KUKA KRL program: MyProgram_208().src

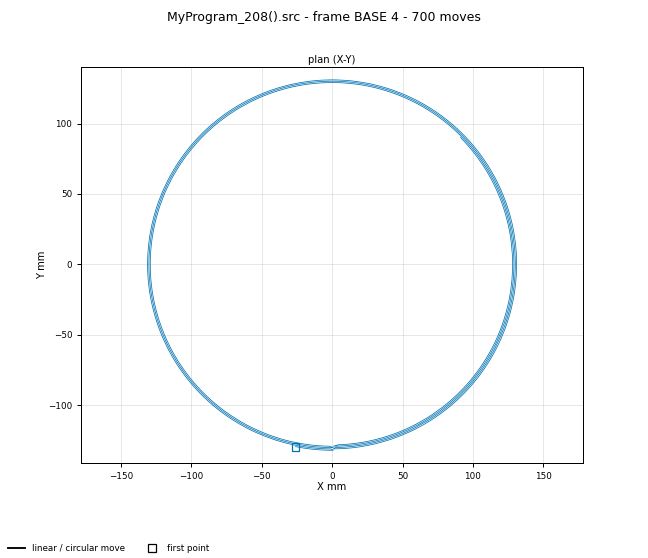
[picture p0: tool path of MyProgram_208().src in frame BASE 4, 700 of 700 moves have a stored position in this frame; points joined in program order, loops and branches not executed]
&ACCESS RVP
&REL 1
&PARAM TEMPLATE = C:\KRC\Roboter\Template\vorgabe
&PARAM EDITMASK = *
DEF MyProgram_208()
; ---- Setting reference (Base) ----
$BASE = BASE_DATA[4]

; --------------------------
; ---- Setting tool (TCP) ----
$TOOL = TOOL_DATA[3]
; --------------------------

$VEL.CP = VEL_APROX_PRINT
Startdeposition()
$VEL.CP = VEL_PRINT
LIN {X -25.9826,Y -129.3712,Z 148,A -104.0355,B 24.9663,C -1.3419,E1 24.9702,E2 190.502} C_DIS
LIN {X -21.9988,Y -130.1078,Z 148,A -102.3686,B 24.9665,C -1.3366,E1 24.9747,E2 188.8461} C_DIS
LIN {X -18.4843,Y -130.6533,Z 148,A -100.8231,B 24.9665,C -1.3362,E1 24.979,E2 187.3001} C_DIS
LIN {X -14.4168,Y -131.1647,Z 148,A -99.072,B 24.9666,C -1.3344,E1 24.9838,E2 185.5521} C_DIS
LIN {X -11.0414,Y -131.4916,Z 148,A -97.5626,B 24.9666,C -1.3363,E1 24.988,E2 184.0376} C_DIS
LIN {X -6.8374,Y -131.7773,Z 148,A -95.7546,B 24.9666,C -1.3352,E1 24.9931,E2 182.2315} C_DIS
LIN {X -3.1641,Y -131.9174,Z 148,A -94.0531,B 24.9663,C -1.3409,E1 24.9979,E2 180.5163} C_DIS
LIN {X 0.9361,Y -131.9509,Z 148,A -93.0717,B 24.9684,C -1.2997,E1 25.0004,E2 179.6325} C_DIS
Enddeposition()
LIN {X 0.9361,Y -131.9509,Z 148,A -93.0717,B 24.9684,C -1.2997,E1 25.0004,E2 179.6325} C_DIS
Startdeposition()
$VEL.CP = VEL_PRINT
LIN {X -0.9099,Y -130.9994,Z 148,A -93.7427,B 24.7462,C -1.2766,E1 24.7754,E2 180.3292} C_DIS
LIN {X -4.2416,Y -130.9351,Z 148,A -95.3676,B 24.7466,C -1.2679,E1 24.7708,E2 181.9751} C_DIS
LIN {X -8.0621,Y -130.754,Z 148,A -96.9489,B 24.7464,C -1.2724,E1 24.7664,E2 183.546} C_DIS
LIN {X -11.7713,Y -130.4745,Z 148,A -98.5272,B 24.7463,C -1.2749,E1 24.7621,E2 185.1191} C_DIS
LIN {X -15.6524,Y -130.0639,Z 148,A -100.2514,B 24.7463,C -1.2743,E1 24.7573,E2 186.8457} C_DIS
LIN {X -18.8652,Y -129.6372,Z 148,A -101.6954,B 24.7463,C -1.2733,E1 24.7533,E2 188.2933} C_DIS
LIN {X -23.4306,Y -128.8903,Z 148,A -103.7209,B 24.7463,C -1.2739,E1 24.7477,E2 190.3196} C_DIS
LIN {X -26.5584,Y -128.2825,Z 148,A -105.065,B 24.7462,C -1.2769,E1 24.744,E2 191.6579} C_DIS
LIN {X -29.9352,Y -127.5384,Z 148,A -106.5997,B 24.7462,C -1.2765,E1 24.7398,E2 193.1955} C_DIS
LIN {X -32.6648,Y -126.8651,Z 148,A -107.8332,B 24.7462,C -1.2771,E1 24.7365,E2 194.4294} C_DIS
LIN {X -35.721,Y -126.0387,Z 148,A -109.2219,B 24.7462,C -1.2778,E1 24.7328,E2 195.8187} C_DIS
LIN {X -38.4449,Y -125.2339,Z 148,A -110.4824,B 24.7462,C -1.2778,E1 24.7294,E2 197.0813} C_DIS
LIN {X -41.7109,Y -124.1847,Z 148,A -111.9951,B 24.7462,C -1.2784,E1 24.7254,E2 198.5953} C_DIS
LIN {X -44.8677,Y -123.0797,Z 148,A -113.4445,B 24.746,C -1.2804,E1 24.7216,E2 200.0429} C_DIS
LIN {X -47.7748,Y -121.9803,Z 148,A -114.8123,B 24.746,C -1.2813,E1 24.718,E2 201.4115} C_DIS
LIN {X -51.0457,Y -120.6491,Z 148,A -116.3473,B 24.7459,C -1.2833,E1 24.714,E2 202.9451} C_DIS
LIN {X -53.8492,Y -119.4232,Z 148,A -117.6982,B 24.7459,C -1.2842,E1 24.7106,E2 204.2971} C_DIS
LIN {X -56.7591,Y -118.0677,Z 148,A -119.1224,B 24.7458,C -1.2849,E1 24.707,E2 205.7232} C_DIS
LIN {X -59.8552,Y -116.5292,Z 148,A -120.6231,B 24.7457,C -1.2874,E1 24.7032,E2 207.2221} C_DIS
LIN {X -62.9418,Y -114.8929,Z 148,A -122.1788,B 24.7457,C -1.2881,E1 24.6994,E2 208.7805} C_DIS
LIN {X -66.1217,Y -113.0928,Z 148,A -123.8872,B 24.7457,C -1.285,E1 24.6953,E2 210.5014} C_DIS
LIN {X -70.1036,Y -110.6685,Z 148,A -125.8821,B 24.7455,C -1.2903,E1 24.6905,E2 212.4899} C_DIS
LIN {X -73.782,Y -108.2515,Z 148,A -127.8213,B 24.7455,C -1.2928,E1 24.686,E2 214.4298} C_DIS
LIN {X -77.2207,Y -105.8259,Z 148,A -129.6872,B 24.7453,C -1.2948,E1 24.6818,E2 216.2975} C_DIS
LIN {X -80.6432,Y -103.2414,Z 148,A -131.5951,B 24.7453,C -1.2966,E1 24.6776,E2 218.2079} C_DIS
LIN {X -84.0166,Y -100.515,Z 148,A -133.4733,B 24.745,C -1.3012,E1 24.6735,E2 220.0824} C_DIS
LIN {X -87.2683,Y -97.705,Z 148,A -135.3719,B 24.7449,C -1.304,E1 24.6695,E2 221.9817} C_DIS
LIN {X -90.6534,Y -94.5727,Z 148,A -137.3709,B 24.7446,C -1.3091,E1 24.6655,E2 223.9768} C_DIS
LIN {X -93.6988,Y -91.5564,Z 148,A -139.1989,B 24.7443,C -1.3154,E1 24.6619,E2 225.7975} C_DIS
LIN {X -96.2825,Y -88.8354,Z 148,A -140.9202,B 24.7443,C -1.3153,E1 24.6586,E2 227.5267} C_DIS
LIN {X -98.9862,Y -85.8131,Z 148,A -142.7358,B 24.7442,C -1.3174,E1 24.6552,E2 229.3455} C_DIS
LIN {X -101.8189,Y -82.4315,Z 148,A -144.6409,B 24.7439,C -1.3232,E1 24.6519,E2 231.2456} C_DIS
LIN {X -104.4895,Y -79.0187,Z 148,A -146.5452,B 24.7437,C -1.3275,E1 24.6486,E2 233.1489} C_DIS
LIN {X -107.1639,Y -75.352,Z 148,A -148.5233,B 24.7434,C -1.3328,E1 24.6454,E2 235.1238} C_DIS
LIN {X -109.6501,Y -71.6869,Z 148,A -150.5262,B 24.7434,C -1.3348,E1 24.6423,E2 237.1321} C_DIS
LIN {X -111.9772,Y -67.9938,Z 148,A -152.4303,B 24.743,C -1.3401,E1 24.6395,E2 239.0332} C_DIS
LIN {X -114.2442,Y -64.1113,Z 148,A -154.3647,B 24.7427,C -1.347,E1 24.6368,E2 240.9611} C_DIS
LIN {X -116.3464,Y -60.213,Z 148,A -156.2318,B 24.7422,C -1.3558,E1 24.6344,E2 242.8173} C_DIS
LIN {X -117.7191,Y -57.4802,Z 148,A -157.5744,B 24.7421,C -1.3594,E1 24.6327,E2 244.1586} C_DIS
LIN {X -119.1027,Y -54.555,Z 148,A -158.9968,B 24.7419,C -1.3631,E1 24.6311,E2 245.5798} C_DIS
LIN {X -120.3978,Y -51.6334,Z 148,A -160.4149,B 24.7417,C -1.3663,E1 24.6295,E2 246.9983} C_DIS
LIN {X -121.6766,Y -48.5441,Z 148,A -161.8738,B 24.7415,C -1.3708,E1 24.6279,E2 248.4546} C_DIS
LIN {X -122.8151,Y -45.5864,Z 148,A -163.2705,B 24.7413,C -1.3744,E1 24.6266,E2 249.8505} C_DIS
LIN {X -123.9258,Y -42.4751,Z 148,A -164.6967,B 24.741,C -1.3797,E1 24.6252,E2 251.2723} C_DIS
LIN {X -124.9291,Y -39.4266,Z 148,A -166.1227,B 24.7408,C -1.3829,E1 24.624,E2 252.6987} C_DIS
LIN {X -125.7713,Y -36.6488,Z 148,A -167.4085,B 24.7407,C -1.3861,E1 24.623,E2 253.9843} C_DIS
LIN {X -126.592,Y -33.7048,Z 148,A -168.7593,B 24.7405,C -1.3896,E1 24.622,E2 255.3347} C_DIS
LIN {X -127.3797,Y -30.5936,Z 148,A -170.171,B 24.7403,C -1.3936,E1 24.6211,E2 256.745} C_DIS
LIN {X -128.107,Y -27.3901,Z 148,A -171.6235,B 24.7401,C -1.3975,E1 24.6202,E2 258.1969} C_DIS
LIN {X -128.7553,Y -24.1625,Z 148,A -173.1573,B 24.7401,C -1.3976,E1 24.6194,E2 259.7394} C_DIS
LIN {X -129.4372,Y -20.1891,Z 148,A -174.8662,B 24.7396,C -1.4059,E1 24.6186,E2 261.4389} C_DIS
LIN {X -129.923,Y -16.7824,Z 148,A -176.3647,B 24.7394,C -1.411,E1 24.618,E2 262.9341} C_DIS
LIN {X -130.331,Y -13.2664,Z 148,A -177.8982,B 24.739,C -1.4167,E1 24.6176,E2 264.4631} C_DIS
LIN {X -130.5736,Y -10.5988,Z 148,A -179.0975,B 24.739,C -1.4192,E1 24.6173,E2 265.6636} C_DIS
LIN {X -130.8584,Y -6.1548,Z 148,A 178.9451,B 24.7386,C -1.4252,E1 24.617,E2 267.6187} C_DIS
LIN {X -130.9711,Y -2.9451,Z 148,A 177.3953,B 24.7387,C -1.423,E1 24.6168,E2 269.1831} C_DIS
LIN {X -131.002,Y 0.7144,Z 148,A 175.8358,B 24.7383,C -1.4302,E1 24.6168,E2 270.7349} C_DIS
LIN {X -130.9337,Y 4.2929,Z 148,A 174.3806,B 24.7378,C -1.4404,E1 24.6169,E2 272.1742} C_DIS
LIN {X -130.8001,Y 7.3151,Z 148,A 173.0287,B 24.7376,C -1.4434,E1 24.6171,E2 273.5272} C_DIS
LIN {X -130.6235,Y 9.9641,Z 148,A 171.835,B 24.7375,C -1.4458,E1 24.6174,E2 274.7225} C_DIS
LIN {X -130.3616,Y 12.9475,Z 148,A 170.5349,B 24.7372,C -1.4506,E1 24.6177,E2 276.0189} C_DIS
LIN {X -129.9903,Y 16.2694,Z 148,A 169.0609,B 24.737,C -1.4548,E1 24.6182,E2 277.4918} C_DIS
LIN {X -129.6518,Y 18.7633,Z 148,A 167.8956,B 24.737,C -1.4554,E1 24.6186,E2 278.6625} C_DIS
LIN {X -129.0893,Y 22.3185,Z 148,A 166.3617,B 24.7366,C -1.4624,E1 24.6193,E2 280.1888} C_DIS
LIN {X -128.5265,Y 25.3597,Z 148,A 164.9976,B 24.7363,C -1.4663,E1 24.62,E2 281.5517} C_DIS
LIN {X -127.9573,Y 28.0834,Z 148,A 163.7659,B 24.7362,C -1.4696,E1 24.6208,E2 282.7828} C_DIS
LIN {X -127.2826,Y 30.9963,Z 148,A 162.4348,B 24.736,C -1.4728,E1 24.6216,E2 284.1141} C_DIS
LIN {X -126.4618,Y 34.1929,Z 148,A 160.9953,B 24.7357,C -1.4776,E1 24.6226,E2 285.5505} C_DIS
LIN {X -125.6529,Y 37.0533,Z 148,A 159.6666,B 24.7355,C -1.4805,E1 24.6237,E2 286.8801} C_DIS
LIN {X -124.7469,Y 39.9969,Z 148,A 158.3113,B 24.7353,C -1.4844,E1 24.6248,E2 288.2338} C_DIS
LIN {X -123.666,Y 43.2244,Z 148,A 156.8135,B 24.7351,C -1.4887,E1 24.6262,E2 289.7299} C_DIS
LIN {X -122.5921,Y 46.1816,Z 148,A 155.4164,B 24.7349,C -1.4921,E1 24.6275,E2 291.1269} C_DIS
LIN {X -121.1977,Y 49.732,Z 148,A 153.7572,B 24.7346,C -1.4977,E1 24.6292,E2 292.782} C_DIS
LIN {X -120.0733,Y 52.384,Z 148,A 152.4837,B 24.7344,C -1.501,E1 24.6306,E2 294.0546} C_DIS
LIN {X -118.56,Y 55.7287,Z 148,A 150.8699,B 24.7341,C -1.5055,E1 24.6325,E2 295.6666} C_DIS
LIN {X -117.3472,Y 58.2341,Z 148,A 149.5948,B 24.7341,C -1.5066,E1 24.6341,E2 296.946} C_DIS
LIN {X -115.263,Y 62.2618,Z 148,A 147.5835,B 24.7338,C -1.5112,E1 24.6367,E2 298.9571} C_DIS
LIN {X -113.1673,Y 65.9948,Z 148,A 145.6202,B 24.7338,C -1.5125,E1 24.6394,E2 300.9276} C_DIS
LIN {X -110.9102,Y 69.7206,Z 148,A 143.7212,B 24.7334,C -1.5183,E1 24.6422,E2 302.8225} C_DIS
LIN {X -108.5273,Y 73.3745,Z 148,A 141.8388,B 24.733,C -1.5249,E1 24.6451,E2 304.6984} C_DIS
LIN {X -105.9314,Y 77.0752,Z 148,A 139.8594,B 24.7327,C -1.5303,E1 24.6483,E2 306.6746} C_DIS
LIN {X -103.3053,Y 80.5614,Z 148,A 137.9087,B 24.7325,C -1.5336,E1 24.6516,E2 308.6269} C_DIS
LIN {X -100.5874,Y 83.9302,Z 148,A 135.9813,B 24.7323,C -1.537,E1 24.655,E2 310.555} C_DIS
LIN {X -97.988,Y 86.9505,Z 148,A 134.3289,B 24.7318,C -1.5458,E1 24.6581,E2 312.1939} C_DIS
LIN {X -95.4585,Y 89.7203,Z 148,A 132.6064,B 24.7318,C -1.5461,E1 24.6613,E2 313.9232} C_DIS
LIN {X -92.6341,Y 92.6341,Z 148,A 130.8693,B 24.7314,C -1.5523,E1 24.6647,E2 315.653} C_DIS
LIN {X -89.7203,Y 95.4585,Z 148,A 129.1108,B 24.7311,C -1.5574,E1 24.6683,E2 317.4067} C_DIS
LIN {X -86.6644,Y 98.241,Z 148,A 127.2293,B 24.7311,C -1.5581,E1 24.6722,E2 319.294} C_DIS
LIN {X -83.3657,Y 101.0555,Z 148,A 125.3837,B 24.7307,C -1.5648,E1 24.6761,E2 321.1307} C_DIS
LIN {X -80.063,Y 103.6917,Z 148,A 123.5555,B 24.7304,C -1.5698,E1 24.6801,E2 322.9537} C_DIS
LIN {X -77.0752,Y 105.9314,Z 148,A 121.8208,B 24.7304,C -1.5685,E1 24.684,E2 324.6979} C_DIS
LIN {X -73.6336,Y 108.3519,Z 148,A 119.9486,B 24.7304,C -1.5707,E1 24.6883,E2 326.5713} C_DIS
LIN {X -69.7206,Y 110.9102,Z 148,A 117.9462,B 24.73,C -1.5767,E1 24.693,E2 328.5658} C_DIS
LIN {X -66.0255,Y 113.1493,Z 148,A 116.0341,B 24.7298,C -1.5791,E1 24.6976,E2 330.478} C_DIS
LIN {X -62.3681,Y 115.2059,Z 148,A 114.1343,B 24.7298,C -1.5792,E1 24.7023,E2 332.383} C_DIS
LIN {X -59.0536,Y 116.9373,Z 148,A 112.6504,B 24.7292,C -1.5892,E1 24.7059,E2 333.8468} C_DIS
LIN {X -55.9395,Y 118.4593,Z 148,A 111.127,B 24.7291,C -1.5913,E1 24.7097,E2 335.3693} C_DIS
LIN {X -52.7398,Y 119.9194,Z 148,A 109.5781,B 24.729,C -1.5931,E1 24.7137,E2 336.9176} C_DIS
LIN {X -50.0533,Y 121.0636,Z 148,A 108.3172,B 24.7288,C -1.5958,E1 24.7169,E2 338.1751} C_DIS
LIN {X -47.1892,Y 122.2079,Z 148,A 106.9282,B 24.7288,C -1.5958,E1 24.7205,E2 339.5672} C_DIS
LIN {X -43.6723,Y 123.5107,Z 148,A 105.3041,B 24.7287,C -1.5986,E1 24.7248,E2 341.1878} C_DIS
LIN {X -40.6267,Y 124.5457,Z 148,A 103.8953,B 24.7286,C -1.6002,E1 24.7285,E2 342.5954} C_DIS
LIN {X -38.1676,Y 125.3188,Z 148,A 102.7699,B 24.7285,C -1.6017,E1 24.7315,E2 343.7192} C_DIS
LIN {X -35.1038,Y 126.2113,Z 148,A 101.3643,B 24.7285,C -1.6027,E1 24.7353,E2 345.1247} C_DIS
LIN {X -32.0077,Y 127.0319,Z 148,A 99.9579,B 24.7283,C -1.6039,E1 24.7391,E2 346.5303} C_DIS
LIN {X -28.7342,Y 127.8127,Z 148,A 98.5168,B 24.7282,C -1.6067,E1 24.743,E2 347.9665} C_DIS
LIN {X -25.3597,Y 128.5265,Z 148,A 96.986,B 24.7282,C -1.6069,E1 24.7472,E2 349.4987} C_DIS
LIN {X -22.5439,Y 129.049,Z 148,A 95.7399,B 24.7281,C -1.6082,E1 24.7506,E2 350.7431} C_DIS
LIN {X -19.6104,Y 129.5268,Z 148,A 94.412,B 24.7281,C -1.6077,E1 24.7543,E2 352.0732} C_DIS
LIN {X -16.5908,Y 129.9481,Z 148,A 93.1019,B 24.728,C -1.6097,E1 24.7579,E2 353.3796} C_DIS
LIN {X -14.0238,Y 130.2495,Z 148,A 91.9555,B 24.728,C -1.6096,E1 24.7611,E2 354.527} C_DIS
LIN {X -10.7428,Y 130.5614,Z 148,A 90.4887,B 24.728,C -1.609,E1 24.7652,E2 355.9959} C_DIS
LIN {X -6.8071,Y 130.8256,Z 148,A 88.7518,B 24.728,C -1.6091,E1 24.77,E2 357.7332} C_DIS
LIN {X -3.2198,Y 130.9635,Z 148,A 87.2292,B 24.7278,C -1.6119,E1 24.7742,E2 359.2492} C_DIS
LIN {X -0.4557,Y 131.0019,Z 148,A 85.8758,B 24.7283,C -1.6051,E1 24.7781,E2 360.619} C_DIS
LIN {X 3.6364,Y 130.9519,Z 148,A 84.2162,B 24.7279,C -1.6117,E1 24.7827,E2 362.2624} C_DIS
LIN {X 7.3151,Y 130.8001,Z 148,A 82.6242,B 24.7278,C -1.6127,E1 24.7871,E2 363.8517} C_DIS
LIN {X 10.2809,Y 130.6004,Z 148,A 81.1754,B 24.7283,C -1.6052,E1 24.7912,E2 365.3176} C_DIS
LIN {X 13.9697,Y 130.2553,Z 148,A 79.6586,B 24.728,C -1.6102,E1 24.7953,E2 366.8216} C_DIS
LIN {X 17.7767,Y 129.7927,Z 148,A 78.0192,B 24.7279,C -1.6117,E1 24.7999,E2 368.4561} C_DIS
LIN {X 22.0621,Y 129.1321,Z 148,A 76.1251,B 24.7279,C -1.6112,E1 24.8051,E2 370.3494} C_DIS
LIN {X 24.7907,Y 128.6352,Z 148,A 74.8752,B 24.728,C -1.6089,E1 24.8085,E2 371.6035} C_DIS
LIN {X 28.0834,Y 127.9573,Z 148,A 73.4127,B 24.728,C -1.6085,E1 24.8125,E2 373.0649} C_DIS
LIN {X 31.4626,Y 127.1702,Z 148,A 71.9179,B 24.728,C -1.6087,E1 24.8166,E2 374.557} C_DIS
LIN {X 34.1929,Y 126.4618,Z 148,A 70.7054,B 24.728,C -1.609,E1 24.8198,E2 375.7668} C_DIS
LIN {X 37.0053,Y 125.6669,Z 148,A 69.3938,B 24.7282,C -1.6064,E1 24.8234,E2 377.0824} C_DIS
LIN {X 40.1901,Y 124.6852,Z 148,A 67.9494,B 24.7282,C -1.6059,E1 24.8272,E2 378.5254} C_DIS
LIN {X 43.2147,Y 123.6694,Z 148,A 66.5628,B 24.7282,C -1.6052,E1 24.8309,E2 379.911} C_DIS
LIN {X 46.5227,Y 122.4644,Z 148,A 65.0073,B 24.7284,C -1.6028,E1 24.835,E2 381.4688} C_DIS
LIN {X 49.3702,Y 121.3436,Z 148,A 63.6779,B 24.7284,C -1.6019,E1 24.8384,E2 382.7973} C_DIS
LIN {X 52.7398,Y 119.9194,Z 148,A 62.0809,B 24.7286,C -1.6003,E1 24.8425,E2 384.3944} C_DIS
LIN {X 55.7287,Y 118.56,Z 148,A 60.6472,B 24.7286,C -1.5987,E1 24.8461,E2 385.8283} C_DIS
LIN {X 58.3798,Y 117.2754,Z 148,A 59.3607,B 24.7287,C -1.5971,E1 24.8494,E2 387.1149} C_DIS
LIN {X 61.3241,Y 115.763,Z 148,A 57.8918,B 24.7289,C -1.5941,E1 24.853,E2 388.5869} C_DIS
LIN {X 65.1192,Y 113.673,Z 148,A 55.9562,B 24.7292,C -1.5893,E1 24.8577,E2 390.5283} C_DIS
LIN {X 68.8477,Y 111.4547,Z 148,A 54.062,B 24.7294,C -1.5865,E1 24.8623,E2 392.423} C_DIS
LIN {X 72.3878,Y 109.1887,Z 148,A 52.2524,B 24.7294,C -1.585,E1 24.8665,E2 394.2303} C_DIS
LIN {X 75.8535,Y 106.8102,Z 148,A 50.467,B 24.7295,C -1.5846,E1 24.8706,E2 396.0105} C_DIS
LIN {X 79.0297,Y 104.4811,Z 148,A 48.712,B 24.7298,C -1.5798,E1 24.8745,E2 397.7705} C_DIS
LIN {X 82.2119,Y 101.996,Z 148,A 46.9168,B 24.7301,C -1.5749,E1 24.8785,E2 399.5705} C_DIS
LIN {X 85.6299,Y 99.144,Z 148,A 44.9716,B 24.7303,C -1.5712,E1 24.8826,E2 401.517} C_DIS
LIN {X 88.8354,Y 96.2825,Z 148,A 43.1745,B 24.7303,C -1.5716,E1 24.8863,E2 403.3058} C_DIS
LIN {X 91.6109,Y 93.6454,Z 148,A 41.4111,B 24.7308,C -1.5634,E1 24.8899,E2 405.0814} C_DIS
LIN {X 94.8522,Y 90.3609,Z 148,A 39.4288,B 24.7309,C -1.5608,E1 24.8937,E2 407.0614} C_DIS
LIN {X 97.7478,Y 87.2205,Z 148,A 37.5996,B 24.7311,C -1.5585,E1 24.8972,E2 408.8878} C_DIS
LIN {X 100.515,Y 84.0166,Z 148,A 35.7335,B 24.7314,C -1.5533,E1 24.9005,E2 410.7576} C_DIS
LIN {X 103.1734,Y 80.7298,Z 148,A 33.8816,B 24.7316,C -1.5486,E1 24.9038,E2 412.6119} C_DIS
LIN {X 105.8259,Y 77.2207,Z 148,A 31.917,B 24.732,C -1.5416,E1 24.907,E2 414.5836} C_DIS
LIN {X 108.3519,Y 73.6336,Z 148,A 30.0263,B 24.7322,C -1.5382,E1 24.9101,E2 416.4732} C_DIS
LIN {X 110.9102,Y 69.7206,Z 148,A 28.0434,B 24.7324,C -1.536,E1 24.913,E2 418.4512} C_DIS
LIN {X 113.1673,Y 65.9948,Z 148,A 26.1559,B 24.7326,C -1.5317,E1 24.9157,E2 420.3392} C_DIS
LIN {X 115.2059,Y 62.3681,Z 148,A 24.2716,B 24.7331,C -1.5232,E1 24.9183,E2 422.2337} C_DIS
LIN {X 117.0275,Y 58.8765,Z 148,A 22.6931,B 24.733,C -1.526,E1 24.9203,E2 423.7971} C_DIS
LIN {X 118.56,Y 55.7287,Z 148,A 21.1812,B 24.7332,C -1.5226,E1 24.9221,E2 425.309} C_DIS
LIN {X 119.6843,Y 53.2656,Z 148,A 20.0021,B 24.7333,C -1.5194,E1 24.9235,E2 426.4891} C_DIS
LIN {X 121.0636,Y 50.0533,Z 148,A 18.488,B 24.7335,C -1.5157,E1 24.9251,E2 428.0036} C_DIS
LIN {X 122.2269,Y 47.1405,Z 148,A 17.133,B 24.7337,C -1.5125,E1 24.9265,E2 429.3587} C_DIS
LIN {X 123.3409,Y 44.1432,Z 148,A 15.7214,B 24.734,C -1.5076,E1 24.9278,E2 430.774} C_DIS
LIN {X 124.3201,Y 41.3042,Z 148,A 14.4251,B 24.7342,C -1.5045,E1 24.929,E2 432.0702} C_DIS
LIN {X 125.3157,Y 38.1777,Z 148,A 12.9994,B 24.7344,C -1.5005,E1 24.9302,E2 433.497} C_DIS
LIN {X 126.2072,Y 35.1185,Z 148,A 11.6291,B 24.7346,C -1.4975,E1 24.9312,E2 434.8667} C_DIS
LIN {X 127.0727,Y 31.8469,Z 148,A 10.1551,B 24.7348,C -1.4931,E1 24.9323,E2 436.3425} C_DIS
LIN {X 127.8127,Y 28.7342,Z 148,A 8.7503,B 24.7351,C -1.4884,E1 24.9332,E2 437.7503} C_DIS
LIN {X 128.6645,Y 24.6376,Z 148,A 6.9511,B 24.7353,C -1.4842,E1 24.9341,E2 439.5487} C_DIS
LIN {X 129.2392,Y 21.42,Z 148,A 5.5014,B 24.7357,C -1.4786,E1 24.9348,E2 441.0034} C_DIS
LIN {X 129.7927,Y 17.7767,Z 148,A 3.942,B 24.7357,C -1.4761,E1 24.9355,E2 442.5593} C_DIS
LIN {X 130.106,Y 15.299,Z 148,A 2.8055,B 24.7361,C -1.4702,E1 24.9358,E2 443.7029} C_DIS
LIN {X 130.4745,Y 11.7713,Z 148,A 1.3213,B 24.7362,C -1.4687,E1 24.9362,E2 445.1818} C_DIS
LIN {X 130.7283,Y 8.4797,Z 148,A -0.2002,B 24.7367,C -1.4599,E1 24.9366,E2 446.7154} C_DIS
LIN {X 130.912,Y 4.872,Z 148,A -1.7245,B 24.7368,C -1.4577,E1 24.9367,E2 448.2357} C_DIS
LIN {X 131.002,Y 0.7144,Z 148,A -3.4745,B 24.7369,C -1.4554,E1 24.9368,E2 449.9806} C_DIS
LIN {X 130.9722,Y -2.9078,Z 148,A -5.2225,B 24.7377,C -1.4413,E1 24.9368,E2 451.7515} C_DIS
LIN {X 130.8339,Y -6.6416,Z 148,A -6.7322,B 24.7377,C -1.4426,E1 24.9366,E2 453.249} C_DIS
LIN {X 130.6236,Y -9.9637,Z 148,A -8.1088,B 24.7377,C -1.4421,E1 24.9363,E2 454.6186} C_DIS
LIN {X 130.3684,Y -12.8768,Z 148,A -9.4087,B 24.738,C -1.4367,E1 24.936,E2 455.9235} C_DIS
LIN {X 130.0947,Y -15.394,Z 148,A -10.5205,B 24.7382,C -1.4329,E1 24.9356,E2 457.0379} C_DIS
LIN {X 129.6895,Y -18.4992,Z 148,A -11.8686,B 24.7384,C -1.4295,E1 24.9351,E2 458.3859} C_DIS
LIN {X 129.2136,Y -21.5734,Z 148,A -13.2338,B 24.7386,C -1.4248,E1 24.9345,E2 459.7542} C_DIS
LIN {X 128.6271,Y -24.8331,Z 148,A -14.6845,B 24.7389,C -1.4199,E1 24.9337,E2 461.208} C_DIS
LIN {X 127.9742,Y -28.0053,Z 148,A -16.0595,B 24.739,C -1.4175,E1 24.933,E2 462.5806} C_DIS
LIN {X 127.3166,Y -30.8556,Z 148,A -17.3794,B 24.7393,C -1.4112,E1 24.9321,E2 463.9077} C_DIS
LIN {X 126.4618,Y -34.1929,Z 148,A -18.8401,B 24.7395,C -1.4087,E1 24.9311,E2 465.3657} C_DIS
LIN {X 125.5957,Y -37.2487,Z 148,A -20.2217,B 24.7397,C -1.4047,E1 24.93,E2 466.749} C_DIS
LIN {X 124.5457,Y -40.6267,Z 148,A -21.7601,B 24.7399,C -1.4001,E1 24.9287,E2 468.2894} C_DIS
LIN {X 123.6698,Y -43.2134,Z 148,A -22.9532,B 24.7401,C -1.3964,E1 24.9276,E2 469.4845} C_DIS
LIN {X 122.553,Y -46.2861,Z 148,A -24.4084,B 24.7404,C -1.3905,E1 24.9262,E2 470.9455} C_DIS
LIN {X 121.1977,Y -49.732,Z 148,A -25.9806,B 24.7406,C -1.388,E1 24.9246,E2 472.515} C_DIS
LIN {X 120.1282,Y -52.2569,Z 148,A -27.1936,B 24.7408,C -1.3835,E1 24.9232,E2 473.7318} C_DIS
LIN {X 118.56,Y -55.7287,Z 148,A -28.83,B 24.741,C -1.3799,E1 24.9213,E2 475.3679} C_DIS
LIN {X 117.2754,Y -58.3798,Z 148,A -30.1338,B 24.7412,C -1.3752,E1 24.9197,E2 476.6759} C_DIS
LIN {X 115.2492,Y -62.2875,Z 148,A -32.083,B 24.7416,C -1.3681,E1 24.9171,E2 478.6317} C_DIS
LIN {X 113.1673,Y -65.9948,Z 148,A -34.0125,B 24.7421,C -1.3588,E1 24.9145,E2 480.5731} C_DIS
LIN {X 110.9102,Y -69.7206,Z 148,A -35.8882,B 24.7423,C -1.3548,E1 24.9117,E2 482.4486} C_DIS
LIN {X 108.4477,Y -73.492,Z 148,A -37.7809,B 24.7423,C -1.3533,E1 24.9088,E2 484.3354} C_DIS
LIN {X 105.9314,Y -77.0752,Z 148,A -39.6338,B 24.7425,C -1.3512,E1 24.9058,E2 486.1842} C_DIS
LIN {X 103.9114,Y -79.7776,Z 148,A -41.1238,B 24.7427,C -1.3464,E1 24.9033,E2 487.6785} C_DIS
LIN {X 101.7057,Y -82.5719,Z 148,A -42.7689,B 24.7432,C -1.3374,E1 24.9004,E2 489.3371} C_DIS
LIN {X 98.8753,Y -85.9403,Z 148,A -44.6686,B 24.7434,C -1.3336,E1 24.8969,E2 491.2371} C_DIS
LIN {X 96.037,Y -89.1007,Z 148,A -46.5061,B 24.7436,C -1.3299,E1 24.8935,E2 493.0753} C_DIS
LIN {X 93.2317,Y -92.0327,Z 148,A -48.1771,B 24.7436,C -1.3309,E1 24.8902,E2 494.7366} C_DIS
LIN {X 90.3932,Y -94.8213,Z 148,A -49.9567,B 24.7438,C -1.3246,E1 24.8867,E2 496.5238} C_DIS
LIN {X 87.2205,Y -97.7478,Z 148,A -51.8564,B 24.7441,C -1.3194,E1 24.8827,E2 498.428} C_DIS
LIN {X 84.0166,Y -100.515,Z 148,A -53.6511,B 24.7441,C -1.3182,E1 24.8789,E2 500.2187} C_DIS
LIN {X 80.7537,Y -103.1546,Z 148,A -55.5423,B 24.7445,C -1.3111,E1 24.8748,E2 502.1195} C_DIS
LIN {X 77.2207,Y -105.8259,Z 148,A -57.5105,B 24.7448,C -1.3053,E1 24.8703,E2 504.0944} C_DIS
LIN {X 73.6336,Y -108.3519,Z 148,A -59.4103,B 24.7449,C -1.3024,E1 24.866,E2 505.9946} C_DIS
LIN {X 69.8274,Y -110.8429,Z 148,A -61.3616,B 24.745,C -1.3004,E1 24.8614,E2 507.9441} C_DIS
LIN {X 65.9948,Y -113.1673,Z 148,A -63.36,B 24.7453,C -1.2948,E1 24.8566,E2 509.9499} C_DIS
LIN {X 62.3681,Y -115.2059,Z 148,A -65.1704,B 24.7454,C -1.292,E1 24.8521,E2 511.7615} C_DIS
LIN {X 59.1648,Y -116.8807,Z 148,A -66.6277,B 24.7453,C -1.2958,E1 24.8486,E2 513.2058} C_DIS
LIN {X 55.7287,Y -118.56,Z 148,A -68.2736,B 24.7453,C -1.2944,E1 24.8444,E2 514.8506} C_DIS
LIN {X 52.961,Y -119.8205,Z 148,A -69.5912,B 24.7453,C -1.293,E1 24.8411,E2 516.1682} C_DIS
LIN {X 50.0533,Y -121.0636,Z 148,A -70.9749,B 24.7455,C -1.2909,E1 24.8375,E2 517.5535} C_DIS
LIN {X 47.0313,Y -122.2693,Z 148,A -72.3811,B 24.7455,C -1.2898,E1 24.8338,E2 518.9594} C_DIS
LIN {X 44.1233,Y -123.3481,Z 148,A -73.7456,B 24.7457,C -1.2875,E1 24.8303,E2 520.3263} C_DIS
LIN {X 41.1815,Y -124.361,Z 148,A -75.1282,B 24.7458,C -1.2847,E1 24.8266,E2 521.713} C_DIS
LIN {X 37.5745,Y -125.5003,Z 148,A -76.7467,B 24.7458,C -1.2845,E1 24.8223,E2 523.3289} C_DIS
LIN {X 34.9655,Y -126.25,Z 148,A -77.9362,B 24.7458,C -1.2831,E1 24.8191,E2 524.5198} C_DIS
LIN {X 31.7159,Y -127.106,Z 148,A -79.3886,B 24.7459,C -1.2825,E1 24.8151,E2 525.9715} C_DIS
LIN {X 28.0834,Y -127.9573,Z 148,A -81.0973,B 24.7462,C -1.2769,E1 24.8105,E2 527.691} C_DIS
LIN {X 24.6708,Y -128.6582,Z 148,A -82.5559,B 24.7461,C -1.279,E1 24.8065,E2 529.143} C_DIS
LIN {X 21.4033,Y -129.242,Z 148,A -84.0214,B 24.7461,C -1.2771,E1 24.8024,E2 530.6114} C_DIS
LIN {X 17.7767,Y -129.7927,Z 148,A -85.5848,B 24.7461,C -1.2781,E1 24.7981,E2 532.1711} C_DIS
LIN {X 14.446,Y -130.2041,Z 148,A -87.1273,B 24.7464,C -1.2734,E1 24.7938,E2 533.7236} C_DIS
LIN {X 10.9505,Y -130.5439,Z 148,A -88.6103,B 24.7463,C -1.2753,E1 24.7897,E2 535.2013} C_DIS
LIN {X 7.5386,Y -130.7863,Z 148,A -90.1836,B 24.7465,C -1.2706,E1 24.7853,E2 536.7849} C_DIS
LIN {X 3.6802,Y -130.9507,Z 148,A -91.8016,B 24.7463,C -1.2737,E1 24.7808,E2 538.3952} C_DIS
LIN {X 0.9276,Y -130.9972,Z 148,A -92.5799,B 24.7453,C -1.2951,E1 24.7788,E2 539.1223} C_DIS
Enddeposition()
LIN {X 0.9276,Y -130.9972,Z 148,A -92.5799,B 24.7453,C -1.2951,E1 24.7788,E2 539.1223} C_DIS
Startdeposition()
$VEL.CP = VEL_PRINT
LIN {X 2.2953,Y -130.0302,Z 148,A -91.3636,B 23.7072,C -1.1309,E1 23.737,E2 538.1694} C_DIS
LIN {X 6.6533,Y -129.8801,Z 148,A -89.594,B 23.7075,C -1.1242,E1 23.7419,E2 536.4172} C_DIS
LIN {X 9.7391,Y -129.6854,Z 148,A -88.0412,B 23.707,C -1.1341,E1 23.7462,E2 534.8404} C_DIS
LIN {X 15.3426,Y -129.1421,Z 148,A -85.4485,B 23.7067,C -1.1411,E1 23.7535,E2 532.2323} C_DIS
LIN {X 22.0886,Y -128.1621,Z 148,A -82.6745,B 23.7071,C -1.1319,E1 23.7611,E2 529.4839} C_DIS
LIN {X 24.9925,Y -127.6274,Z 148,A -81.1427,B 23.7066,C -1.1444,E1 23.7654,E2 527.9229} C_DIS
LIN {X 28.6488,Y -126.8557,Z 148,A -79.6943,B 23.7069,C -1.1361,E1 23.7692,E2 526.4972} C_DIS
LIN {X 32.1676,Y -126.0091,Z 148,A -78.1664,B 23.707,C -1.1344,E1 23.7734,E2 524.9759} C_DIS
LIN {X 35.2573,Y -125.1799,Z 148,A -76.7005,B 23.7068,C -1.1387,E1 23.7773,E2 523.5019} C_DIS
LIN {X 40.3053,Y -123.649,Z 148,A -74.4302,B 23.7068,C -1.1387,E1 23.7834,E2 521.2359} C_DIS
LIN {X 42.7685,Y -122.8165,Z 148,A -73.2712,B 23.7068,C -1.1409,E1 23.7864,E2 520.0739} C_DIS
LIN {X 46.2368,Y -121.5549,Z 148,A -71.1381,B 23.7054,C -1.1686,E1 23.7922,E2 517.877} C_DIS
LIN {X 50.1024,Y -120.0114,Z 148,A -69.7611,B 23.7064,C -1.1482,E1 23.7956,E2 516.5539} C_DIS
LIN {X 53.2812,Y -118.6344,Z 148,A -68.2432,B 23.7063,C -1.1501,E1 23.7995,E2 515.0352} C_DIS
LIN {X 56.4292,Y -117.1703,Z 148,A -66.7981,B 23.7063,C -1.1483,E1 23.8031,E2 513.5986} C_DIS
LIN {X 59.5458,Y -115.6185,Z 148,A -65.1445,B 23.706,C -1.1569,E1 23.8073,E2 511.9285} C_DIS
LIN {X 68.4575,Y -110.5763,Z 148,A -60.8352,B 23.706,C -1.1547,E1 23.8177,E2 507.6383} C_DIS
LIN {X 71.6464,Y -108.5371,Z 148,A -59.1404,B 23.7059,C -1.1594,E1 23.8216,E2 505.9379} C_DIS
LIN {X 73.7755,Y -107.1013,Z 148,A -57.8907,B 23.7055,C -1.1677,E1 23.8245,E2 504.6722} C_DIS
LIN {X 77.141,Y -104.7032,Z 148,A -56.0866,B 23.7054,C -1.1706,E1 23.8286,E2 502.8674} C_DIS
LIN {X 80.6325,Y -102.0392,Z 148,A -53.9414,B 23.7047,C -1.1856,E1 23.8334,E2 500.6936} C_DIS
LIN {X 84.5859,Y -98.7868,Z 148,A -51.9149,B 23.705,C -1.179,E1 23.8377,E2 498.6918} C_DIS
LIN {X 87.493,Y -96.2209,Z 148,A -50.2088,B 23.7048,C -1.1829,E1 23.8412,E2 496.9833} C_DIS
LIN {X 90.7138,Y -93.1912,Z 148,A -48.0833,B 23.7041,C -1.1967,E1 23.8456,E2 494.8329} C_DIS
LIN {X 95.3225,Y -88.4711,Z 148,A -45.4695,B 23.7045,C -1.1889,E1 23.8506,E2 492.2504} C_DIS
LIN {X 97.7461,Y -85.7864,Z 148,A -43.7702,B 23.704,C -1.1984,E1 23.8537,E2 490.5355} C_DIS
LIN {X 100.499,Y -82.544,Z 148,A -41.911,B 23.7038,C -1.2026,E1 23.8571,E2 488.6749} C_DIS
LIN {X 104.8446,Y -76.9485,Z 148,A -38.866,B 23.7036,C -1.2072,E1 23.8622,E2 485.634} C_DIS
LIN {X 107.2408,Y -73.5723,Z 148,A -36.9714,B 23.7032,C -1.2159,E1 23.8653,E2 483.7276} C_DIS
LIN {X 109.7634,Y -69.754,Z 148,A -34.9555,B 23.7029,C -1.2216,E1 23.8683,E2 481.7083} C_DIS
LIN {X 112.1721,Y -65.8095,Z 148,A -33.0092,B 23.7029,C -1.2229,E1 23.8711,E2 479.7694} C_DIS
LIN {X 114.3113,Y -62.0199,Z 148,A -31.067,B 23.7025,C -1.2299,E1 23.8738,E2 477.8207} C_DIS
LIN {X 115.9464,Y -58.9017,Z 148,A -28.4624,B 23.6995,C -1.2896,E1 23.8772,E2 475.083} C_DIS
LIN {X 119.1992,Y -52.0068,Z 148,A -25.8254,B 23.7009,C -1.262,E1 23.8801,E2 472.5297} C_DIS
LIN {X 120.7381,Y -48.3258,Z 148,A -24.6417,B 23.7021,C -1.2376,E1 23.8813,E2 471.4132} C_DIS
LIN {X 121.7721,Y -45.6569,Z 148,A -23.3042,B 23.7018,C -1.2455,E1 23.8826,E2 470.0641} C_DIS
LIN {X 122.8587,Y -42.6466,Z 148,A -21.8722,B 23.7015,C -1.2511,E1 23.8839,E2 468.6268} C_DIS
LIN {X 123.9362,Y -39.4062,Z 148,A -20.377,B 23.7013,C -1.2553,E1 23.8852,E2 467.1299} C_DIS
LIN {X 125.1218,Y -35.4647,Z 148,A -18.561,B 23.701,C -1.2613,E1 23.8866,E2 465.3104} C_DIS
LIN {X 126.0203,Y -32.1237,Z 148,A -17.0646,B 23.7008,C -1.2647,E1 23.8877,E2 463.8145} C_DIS
LIN {X 126.8016,Y -28.8859,Z 148,A -15.6363,B 23.7007,C -1.2674,E1 23.8886,E2 462.3884} C_DIS
LIN {X 127.7404,Y -24.4014,Z 148,A -13.5464,B 23.7001,C -1.2776,E1 23.8898,E2 460.2861} C_DIS
LIN {X 128.4897,Y -20.0868,Z 148,A -11.6788,B 23.7,C -1.2807,E1 23.8906,E2 458.4225} C_DIS
LIN {X 128.9973,Y -16.5203,Z 148,A -9.8632,B 23.6991,C -1.2977,E1 23.8913,E2 456.5761} C_DIS
LIN {X 129.5403,Y -11.5212,Z 148,A -7.8346,B 23.6992,C -1.2952,E1 23.8918,E2 454.5665} C_DIS
LIN {X 129.8602,Y -7.0499,Z 148,A -6.0844,B 23.6995,C -1.29,E1 23.8922,E2 452.8402} C_DIS
LIN {X 130.0292,Y -2.3595,Z 148,A -3.7403,B 23.6984,C -1.3111,E1 23.8924,E2 450.4587} C_DIS
LIN {X 130.045,Y 1.3751,Z 148,A -2.3098,B 23.6987,C -1.3053,E1 23.8924,E2 449.0516} C_DIS
LIN {X 129.9651,Y 4.7226,Z 148,A -0.8294,B 23.6985,C -1.3104,E1 23.8922,E2 447.5679} C_DIS
LIN {X 129.7939,Y 8.165,Z 148,A 0.7383,B 23.6981,C -1.3179,E1 23.892,E2 445.9916} C_DIS
LIN {X 129.305,Y 13.9025,Z 148,A 2.8947,B 23.6987,C -1.3064,E1 23.8915,E2 443.8772} C_DIS
LIN {X 128.4526,Y 20.3265,Z 148,A 6.0721,B 23.6973,C -1.3321,E1 23.8902,E2 440.656} C_DIS
LIN {X 127.8429,Y 23.8649,Z 148,A 7.9085,B 23.6963,C -1.3503,E1 23.8893,E2 438.786} C_DIS
LIN {X 127.02,Y 27.9137,Z 148,A 9.4046,B 23.6969,C -1.3392,E1 23.8884,E2 437.3265} C_DIS
LIN {X 126.3945,Y 30.6184,Z 148,A 10.6068,B 23.6968,C -1.342,E1 23.8877,E2 436.1249} C_DIS
LIN {X 125.6331,Y 33.6058,Z 148,A 11.9971,B 23.6965,C -1.3479,E1 23.8867,E2 434.7286} C_DIS
LIN {X 124.5943,Y 37.2809,Z 148,A 13.8105,B 23.6958,C -1.3598,E1 23.8852,E2 432.8968} C_DIS
LIN {X 123.4235,Y 40.9834,Z 148,A 15.3828,B 23.6959,C -1.3579,E1 23.8839,E2 431.3386} C_DIS
LIN {X 122.2954,Y 44.2361,Z 148,A 16.8735,B 23.6958,C -1.3611,E1 23.8825,E2 429.8488} C_DIS
LIN {X 120.9876,Y 47.7008,Z 148,A 19.1439,B 23.6937,C -1.3989,E1 23.8801,E2 427.4984} C_DIS
LIN {X 119.0594,Y 52.3283,Z 148,A 20.6469,B 23.6953,C -1.3689,E1 23.8785,E2 426.0782} C_DIS
LIN {X 117.4073,Y 55.9331,Z 148,A 22.1513,B 23.6957,C -1.3615,E1 23.8768,E2 424.6006} C_DIS
LIN {X 116.527,Y 57.7449,Z 148,A 23.2987,B 23.6949,C -1.3773,E1 23.8753,E2 423.4207} C_DIS
LIN {X 114.9731,Y 60.7806,Z 148,A 24.8278,B 23.6946,C -1.3829,E1 23.8734,E2 421.8864} C_DIS
LIN {X 112.8485,Y 64.6431,Z 148,A 27.4784,B 23.6922,C -1.4246,E1 23.8696,E2 419.1472} C_DIS
LIN {X 110.0125,Y 69.3594,Z 148,A 29.2375,B 23.6938,C -1.3968,E1 23.8671,E2 417.4662} C_DIS
LIN {X 107.5387,Y 73.1366,Z 148,A 31.2003,B 23.6936,C -1.4007,E1 23.8641,E2 415.5043} C_DIS
LIN {X 105.0513,Y 76.6671,Z 148,A 33.1462,B 23.6932,C -1.4077,E1 23.8609,E2 413.551} C_DIS
LIN {X 102.3407,Y 80.2487,Z 148,A 35.0574,B 23.6932,C -1.4091,E1 23.8576,E2 411.6458} C_DIS
LIN {X 99.555,Y 83.6796,Z 148,A 36.9948,B 23.6929,C -1.4133,E1 23.8542,E2 409.7075} C_DIS
LIN {X 96.6473,Y 87.0223,Z 148,A 39.4574,B 23.6912,C -1.4437,E1 23.8495,E2 407.1812} C_DIS
LIN {X 93.4223,Y 90.475,Z 148,A 40.8453,B 23.6929,C -1.4132,E1 23.847,E2 405.8753} C_DIS
LIN {X 90.842,Y 93.0661,Z 148,A 42.9214,B 23.6914,C -1.4401,E1 23.8427,E2 403.7418} C_DIS
LIN {X 88.1871,Y 95.5853,Z 148,A 44.155,B 23.6923,C -1.4243,E1 23.8403,E2 402.5525} C_DIS
LIN {X 85.4811,Y 98.0125,Z 148,A 45.8187,B 23.6919,C -1.4307,E1 23.8368,E2 400.8801} C_DIS
LIN {X 82.0334,Y 100.9163,Z 148,A 47.8151,B 23.6917,C -1.435,E1 23.8325,E2 398.881} C_DIS
LIN {X 78.5567,Y 103.6455,Z 148,A 49.7254,B 23.6916,C -1.4368,E1 23.8283,E2 396.9738} C_DIS
LIN {X 75.1686,Y 106.1283,Z 148,A 51.6047,B 23.6913,C -1.4415,E1 23.824,E2 395.0899} C_DIS
LIN {X 71.4553,Y 108.6628,Z 148,A 53.563,B 23.6912,C -1.4436,E1 23.8195,E2 393.1333} C_DIS
LIN {X 67.6252,Y 111.0875,Z 148,A 55.5833,B 23.6909,C -1.4479,E1 23.8147,E2 391.1092} C_DIS
LIN {X 63.7927,Y 113.3312,Z 148,A 57.4818,B 23.6909,C -1.4479,E1 23.8101,E2 389.2169} C_DIS
LIN {X 59.8603,Y 115.4563,Z 148,A 59.3477,B 23.6911,C -1.4454,E1 23.8055,E2 387.3625} C_DIS
LIN {X 57.4965,Y 116.6495,Z 148,A 60.513,B 23.691,C -1.4469,E1 23.8026,E2 386.1969} C_DIS
LIN {X 54.6446,Y 118.0125,Z 148,A 61.9197,B 23.6908,C -1.4493,E1 23.799,E2 384.7881} C_DIS
LIN {X 51.318,Y 119.497,Z 148,A 63.5134,B 23.6908,C -1.4506,E1 23.7949,E2 383.1954} C_DIS
LIN {X 48.0134,Y 120.8641,Z 148,A 65.3024,B 23.6901,C -1.4627,E1 23.7902,E2 381.3806} C_DIS
LIN {X 44.1092,Y 122.3412,Z 148,A 66.9275,B 23.6906,C -1.4539,E1 23.7861,E2 379.7808} C_DIS
LIN {X 40.9409,Y 123.4377,Z 148,A 68.3859,B 23.6906,C -1.4543,E1 23.7822,E2 378.3245} C_DIS
LIN {X 37.7146,Y 124.4618,Z 148,A 69.9072,B 23.6904,C -1.4569,E1 23.7781,E2 376.7996} C_DIS
LIN {X 33.7301,Y 125.6,Z 148,A 71.7538,B 23.6903,C -1.4592,E1 23.7732,E2 374.9506} C_DIS
LIN {X 29.982,Y 126.5479,Z 148,A 73.3656,B 23.6905,C -1.4558,E1 23.7688,E2 373.3498} C_DIS
LIN {X 27.2776,Y 127.1574,Z 148,A 74.6881,B 23.6901,C -1.4613,E1 23.7652,E2 372.0153} C_DIS
LIN {X 23.1182,Y 127.9791,Z 148,A 77.0053,B 23.6888,C -1.4839,E1 23.7587,E2 369.6448} C_DIS
LIN {X 18.8854,Y 128.6726,Z 148,A 78.4843,B 23.6899,C -1.4646,E1 23.7547,E2 368.2154} C_DIS
LIN {X 14.5056,Y 129.2401,Z 148,A 80.2388,B 23.6905,C -1.4558,E1 23.7499,E2 366.4842} C_DIS
LIN {X 8.07,Y 129.7998,Z 148,A 83.4088,B 23.6895,C -1.4715,E1 23.741,E2 363.2767} C_DIS
LIN {X 4.0818,Y 129.9872,Z 148,A 84.9941,B 23.69,C -1.4631,E1 23.7366,E2 361.7129} C_DIS
LIN {X 0.548,Y 130.0494,Z 148,A 86.5701,B 23.69,C -1.4637,E1 23.7322,E2 360.1354} C_DIS
LIN {X -5.1544,Y 129.9482,Z 148,A 89.0445,B 23.6901,C -1.4612,E1 23.7253,E2 357.6668} C_DIS
LIN {X -11.5584,Y 129.5371,Z 148,A 91.7441,B 23.6906,C -1.454,E1 23.7179,E2 354.9843} C_DIS
LIN {X -15.6756,Y 129.1024,Z 148,A 93.7157,B 23.6902,C -1.46,E1 23.7123,E2 352.9965} C_DIS
LIN {X -21.5546,Y 128.2516,Z 148,A 96.3552,B 23.6902,C -1.4593,E1 23.7051,E2 350.3563} C_DIS
LIN {X -24.9746,Y 127.6309,Z 148,A 97.786,B 23.6906,C -1.4533,E1 23.7012,E2 348.9386} C_DIS
LIN {X -28.4018,Y 126.9122,Z 148,A 99.4538,B 23.6903,C -1.4578,E1 23.6966,E2 347.2574} C_DIS
LIN {X -32.0276,Y 126.0447,Z 148,A 101.0035,B 23.6907,C -1.4519,E1 23.6924,E2 345.7202} C_DIS
LIN {X -35.2536,Y 125.1809,Z 148,A 102.4787,B 23.6907,C -1.4506,E1 23.6884,E2 344.2459} C_DIS
LIN {X -38.4131,Y 124.248,Z 148,A 104.2828,B 23.6899,C -1.4654,E1 23.6835,E2 342.4015} C_DIS
LIN {X -41.6499,Y 123.201,Z 148,A 105.4677,B 23.6909,C -1.449,E1 23.6805,E2 341.2553} C_DIS
LIN {X -45.8053,Y 121.7165,Z 148,A 107.3919,B 23.691,C -1.4456,E1 23.6755,E2 339.3355} C_DIS
LIN {X -48.989,Y 120.4708,Z 148,A 108.9911,B 23.691,C -1.4478,E1 23.6713,E2 337.727} C_DIS
LIN {X -52.3437,Y 119.0533,Z 148,A 110.5262,B 23.6912,C -1.4422,E1 23.6674,E2 336.202} C_DIS
LIN {X -54.7437,Y 117.9666,Z 148,A 111.6662,B 23.6914,C -1.4395,E1 23.6645,E2 335.0658} C_DIS
LIN {X -57.6898,Y 116.5542,Z 148,A 113.0943,B 23.6916,C -1.4367,E1 23.6609,E2 333.6407} C_DIS
LIN {X -60.5395,Y 115.0997,Z 148,A 114.9567,B 23.6905,C -1.4553,E1 23.6562,E2 331.7266} C_DIS
LIN {X -63.9869,Y 113.2221,Z 148,A 116.3126,B 23.6917,C -1.435,E1 23.653,E2 330.4172} C_DIS
LIN {X -68.1466,Y 110.7679,Z 148,A 118.4412,B 23.6919,C -1.4311,E1 23.6479,E2 328.2912} C_DIS
LIN {X -71.4965,Y 108.6357,Z 148,A 120.2839,B 23.6919,C -1.432,E1 23.6436,E2 326.44} C_DIS
LIN {X -74.9043,Y 106.3147,Z 148,A 122.0289,B 23.6922,C -1.4251,E1 23.6396,E2 324.7059} C_DIS
LIN {X -77.9963,Y 104.068,Z 148,A 123.7349,B 23.6924,C -1.4226,E1 23.6357,E2 322.9998} C_DIS
LIN {X -81.1361,Y 101.6387,Z 148,A 125.4443,B 23.6927,C -1.417,E1 23.632,E2 321.2977} C_DIS
LIN {X -84.9157,Y 98.5028,Z 148,A 127.8378,B 23.6924,C -1.4226,E1 23.6269,E2 318.8803} C_DIS
LIN {X -87.8046,Y 95.9369,Z 148,A 129.4052,B 23.6929,C -1.4125,E1 23.6236,E2 317.3315} C_DIS
LIN {X -90.8784,Y 93.0304,Z 148,A 131.2515,B 23.6932,C -1.4073,E1 23.6199,E2 315.4902} C_DIS
LIN {X -93.6002,Y 90.2913,Z 148,A 132.9653,B 23.6934,C -1.4037,E1 23.6166,E2 313.7775} C_DIS
LIN {X -96.2653,Y 87.4441,Z 148,A 134.7161,B 23.6936,C -1.4008,E1 23.6133,E2 312.0257} C_DIS
LIN {X -99.0929,Y 84.2262,Z 148,A 136.5799,B 23.6939,C -1.3949,E1 23.6099,E2 310.1678} C_DIS
LIN {X -101.7753,Y 80.9646,Z 148,A 138.4813,B 23.6941,C -1.3918,E1 23.6065,E2 308.2647} C_DIS
LIN {X -104.4751,Y 77.4499,Z 148,A 140.5231,B 23.6941,C -1.3906,E1 23.6031,E2 306.2157} C_DIS
LIN {X -107.0781,Y 73.8093,Z 148,A 142.4548,B 23.6946,C -1.3833,E1 23.6,E2 304.2921} C_DIS
LIN {X -109.376,Y 70.3594,Z 148,A 144.321,B 23.6947,C -1.3799,E1 23.5972,E2 302.4244} C_DIS
LIN {X -112.3088,Y 65.5768,Z 148,A 146.7066,B 23.6953,C -1.3689,E1 23.5937,E2 300.0532} C_DIS
LIN {X -114.3423,Y 61.9631,Z 148,A 148.6641,B 23.6953,C -1.3694,E1 23.5911,E2 298.0836} C_DIS
LIN {X -116.4348,Y 57.9319,Z 148,A 150.8654,B 23.6951,C -1.3725,E1 23.5883,E2 295.8622} C_DIS
LIN {X -117.8692,Y 54.9543,Z 148,A 151.8369,B 23.6966,C -1.3464,E1 23.5872,E2 294.9503} C_DIS
LIN {X -119.523,Y 51.2581,Z 148,A 153.812,B 23.6964,C -1.3494,E1 23.585,E2 292.956} C_DIS
LIN {X -121.2267,Y 47.0858,Z 148,A 155.8057,B 23.6967,C -1.3437,E1 23.5829,E2 290.9649} C_DIS
LIN {X -122.3442,Y 44.101,Z 148,A 157.1988,B 23.697,C -1.3388,E1 23.5816,E2 289.5757} C_DIS
LIN {X -123.4101,Y 41.0239,Z 148,A 158.6749,B 23.6971,C -1.3361,E1 23.5802,E2 288.0974} C_DIS
LIN {X -124.441,Y 37.7826,Z 148,A 160.4475,B 23.6967,C -1.3436,E1 23.5787,E2 286.2951} C_DIS
LIN {X -125.6321,Y 33.6097,Z 148,A 162.0908,B 23.6977,C -1.3255,E1 23.5776,E2 284.6869} C_DIS
LIN {X -126.4616,Y 30.34,Z 148,A 163.6242,B 23.6978,C -1.3229,E1 23.5765,E2 283.1507} C_DIS
LIN {X -127.2226,Y 26.9756,Z 148,A 165.0693,B 23.6982,C -1.3147,E1 23.5757,E2 281.7171} C_DIS
LIN {X -127.7981,Y 24.0998,Z 148,A 166.5203,B 23.6981,C -1.3176,E1 23.5749,E2 280.2498} C_DIS
LIN {X -128.5061,Y 19.9812,Z 148,A 168.2875,B 23.6986,C -1.3083,E1 23.5741,E2 278.4946} C_DIS
LIN {X -129.047,Y 16.1397,Z 148,A 169.9626,B 23.6989,C -1.3012,E1 23.5735,E2 276.8267} C_DIS
LIN {X -129.3512,Y 13.4737,Z 148,A 171.1324,B 23.6992,C -1.2968,E1 23.5731,E2 275.6604} C_DIS
LIN {X -129.5945,Y 10.8794,Z 148,A 172.3656,B 23.6992,C -1.2969,E1 23.5728,E2 274.4191} C_DIS
LIN {X -129.8717,Y 6.8206,Z 148,A 174.206,B 23.6993,C -1.2932,E1 23.5725,E2 272.5763} C_DIS
LIN {X -130.0196,Y 2.9141,Z 148,A 176.1031,B 23.6993,C -1.2954,E1 23.5724,E2 270.6616} C_DIS
LIN {X -130.0361,Y -1.9427,Z 148,A 177.9413,B 23.7003,C -1.275,E1 23.5724,E2 268.8627} C_DIS
LIN {X -129.9616,Y -4.8127,Z 148,A 179.3408,B 23.7002,C -1.2769,E1 23.5725,E2 267.4495} C_DIS
LIN {X -129.7694,Y -8.5619,Z 148,A -178.8792,B 23.7002,C -1.2771,E1 23.5728,E2 265.6575} C_DIS
LIN {X -129.4244,Y -12.7484,Z 148,A -177.2271,B 23.7009,C -1.2623,E1 23.5732,E2 264.032} C_DIS
LIN {X -129.1226,Y -15.5064,Z 148,A -175.9007,B 23.7009,C -1.2631,E1 23.5737,E2 262.6953} C_DIS
LIN {X -128.5628,Y -19.6152,Z 148,A -174.0528,B 23.7011,C -1.2582,E1 23.5744,E2 260.8479} C_DIS
LIN {X -127.9889,Y -23.063,Z 148,A -172.5076,B 23.7014,C -1.2535,E1 23.5751,E2 259.3046} C_DIS
LIN {X -127.2113,Y -27.0281,Z 148,A -170.6808,B 23.7015,C -1.25,E1 23.5761,E2 257.4752} C_DIS
LIN {X -126.3944,Y -30.6189,Z 148,A -169.1222,B 23.7019,C -1.2421,E1 23.5771,E2 255.9267} C_DIS
LIN {X -125.5154,Y -34.0472,Z 148,A -167.5916,B 23.7022,C -1.236,E1 23.5782,E2 254.402} C_DIS
LIN {X -124.7457,Y -36.7639,Z 148,A -166.2611,B 23.7022,C -1.236,E1 23.5793,E2 253.0631} C_DIS
LIN {X -123.517,Y -40.7028,Z 148,A -163.9514,B 23.7014,C -1.2527,E1 23.5813,E2 250.6975} C_DIS
LIN {X -122.1211,Y -44.7198,Z 148,A -162.7665,B 23.7032,C -1.216,E1 23.5824,E2 249.5975} C_DIS
LIN {X -120.8885,Y -47.9527,Z 148,A -161.0757,B 23.7031,C -1.219,E1 23.5841,E2 247.8892} C_DIS
LIN {X -119.3468,Y -51.6655,Z 148,A -159.2675,B 23.7032,C -1.2155,E1 23.586,E2 246.079} C_DIS
LIN {X -118.0885,Y -54.4801,Z 148,A -157.8907,B 23.7034,C -1.2125,E1 23.5876,E2 244.7019} C_DIS
LIN {X -116.6762,Y -57.4425,Z 148,A -156.424,B 23.7035,C -1.2093,E1 23.5894,E2 243.2346} C_DIS
LIN {X -115.2082,Y -60.3329,Z 148,A -154.8652,B 23.7035,C -1.2112,E1 23.5914,E2 241.6622} C_DIS
LIN {X -113.0346,Y -64.317,Z 148,A -152.8569,B 23.7037,C -1.2061,E1 23.5941,E2 239.6554} C_DIS
LIN {X -110.6491,Y -68.3404,Z 148,A -150.7664,B 23.7039,C -1.202,E1 23.5972,E2 237.564} C_DIS
LIN {X -108.2577,Y -72.0678,Z 148,A -148.8348,B 23.7042,C -1.196,E1 23.6001,E2 235.6371} C_DIS
LIN {X -105.6664,Y -75.8164,Z 148,A -146.8556,B 23.7045,C -1.1896,E1 23.6033,E2 233.6636} C_DIS
LIN {X -103.0925,Y -79.2812,Z 148,A -144.7876,B 23.7043,C -1.1925,E1 23.6068,E2 231.5777} C_DIS
LIN {X -99.9084,Y -83.2582,Z 148,A -142.6328,B 23.7048,C -1.183,E1 23.6106,E2 229.436} C_DIS
LIN {X -97.2544,Y -86.343,Z 148,A -140.8579,B 23.705,C -1.1781,E1 23.6139,E2 227.665} C_DIS
LIN {X -94.3439,Y -89.5144,Z 148,A -138.9229,B 23.7051,C -1.1756,E1 23.6175,E2 225.7271} C_DIS
LIN {X -91.3065,Y -92.6104,Z 148,A -137.0011,B 23.7053,C -1.172,E1 23.6213,E2 223.8057} C_DIS
LIN {X -88.1856,Y -95.5867,Z 148,A -135.0973,B 23.7055,C -1.1683,E1 23.6252,E2 221.903} C_DIS
LIN {X -84.8425,Y -98.5658,Z 148,A -133.1337,B 23.7057,C -1.1639,E1 23.6293,E2 219.942} C_DIS
LIN {X -81.3721,Y -101.4503,Z 148,A -131.105,B 23.7057,C -1.1621,E1 23.6337,E2 217.9099} C_DIS
LIN {X -77.8712,Y -104.1615,Z 148,A -129.1803,B 23.706,C -1.1573,E1 23.638,E2 215.9896} C_DIS
LIN {X -74.0474,Y -106.9136,Z 148,A -127.3549,B 23.7067,C -1.1421,E1 23.6421,E2 214.1954} C_DIS
LIN {X -71.6467,Y -108.5368,Z 148,A -125.8061,B 23.7062,C -1.1528,E1 23.6458,E2 212.6147} C_DIS
LIN {X -67.9743,Y -110.8736,Z 148,A -123.8443,B 23.7062,C -1.1519,E1 23.6504,E2 210.6485} C_DIS
LIN {X -63.9674,Y -113.2331,Z 148,A -121.8295,B 23.7064,C -1.1473,E1 23.6553,E2 208.6387} C_DIS
LIN {X -60.4001,Y -115.1729,Z 148,A -120.1192,B 23.7067,C -1.1413,E1 23.6595,E2 206.9385} C_DIS
LIN {X -57.2748,Y -116.7589,Z 148,A -118.5832,B 23.7068,C -1.139,E1 23.6633,E2 205.404} C_DIS
LIN {X -53.4893,Y -118.5413,Z 148,A -116.8662,B 23.7072,C -1.1308,E1 23.6676,E2 203.7027} C_DIS
LIN {X -50.3544,Y -119.9061,Z 148,A -115.099,B 23.7067,C -1.1415,E1 23.6722,E2 201.9044} C_DIS
LIN {X -45.945,Y -121.6642,Z 148,A -113.0928,B 23.707,C -1.1355,E1 23.6774,E2 199.9089} C_DIS
LIN {X -42.6421,Y -122.8603,Z 148,A -111.584,B 23.7071,C -1.1323,E1 23.6814,E2 198.4049} C_DIS
LIN {X -39.5354,Y -123.8949,Z 148,A -110.1441,B 23.7071,C -1.131,E1 23.6852,E2 196.9654} C_DIS
LIN {X -36.2683,Y -124.8908,Z 148,A -108.5129,B 23.7069,C -1.1359,E1 23.6896,E2 195.3189} C_DIS
LIN {X -32.332,Y -125.9674,Z 148,A -106.7962,B 23.7072,C -1.1309,E1 23.6942,E2 193.612} C_DIS
LIN {X -28.7451,Y -126.8337,Z 148,A -105.1813,B 23.7072,C -1.1296,E1 23.6986,E2 191.9983} C_DIS
LIN {X -22.9401,Y -128.0109,Z 148,A -102.8068,B 23.7078,C -1.1172,E1 23.7051,E2 189.6517} C_DIS
LIN {X -18.6648,Y -128.7042,Z 148,A -100.907,B 23.7078,C -1.1162,E1 23.7103,E2 187.7527} C_DIS
LIN {X -16.649,Y -128.9804,Z 148,A -99.7395,B 23.7073,C -1.1291,E1 23.7136,E2 186.5522} C_DIS
LIN {X -11.6207,Y -129.5317,Z 148,A -97.3706,B 23.707,C -1.1356,E1 23.7202,E2 184.1655} C_DIS
LIN {X -7.6347,Y -129.8266,Z 148,A -95.6809,B 23.7071,C -1.1322,E1 23.7249,E2 182.4838} C_DIS
LIN {X -3.5403,Y -130.0022,Z 148,A -93.9696,B 23.7073,C -1.1278,E1 23.7297,E2 180.783} C_DIS
LIN {X 0.9287,Y -130.0452,Z 148,A -92.7812,B 23.709,C -1.0904,E1 23.7328,E2 179.6877} C_DIS
Enddeposition()
LIN {X 0.9287,Y -130.0452,Z 148,A -92.7812,B 23.709,C -1.0904,E1 23.7328,E2 179.6877} C_DIS
Startdeposition()
$VEL.CP = VEL_PRINT
LIN {X -1.8305,Y -129.0858,Z 148,A -93.6768,B 22.8294,C -0.9549,E1 22.8453,E2 180.8176} C_DIS
LIN {X -6.0098,Y -128.9593,Z 148,A -95.5875,B 22.8295,C -0.9523,E1 22.8399,E2 182.7356} C_DIS
LIN {X -9.9413,Y -128.716,Z 148,A -97.8629,B 22.8304,C -0.9284,E1 22.8334,E2 185.0737} C_DIS
LIN {X -14.6915,Y -128.261,Z 148,A -99.3024,B 22.8292,C -0.9594,E1 22.8296,E2 186.4341} C_DIS
LIN {X -17.7172,Y -127.8778,Z 148,A -101.0063,B 22.8298,C -0.9438,E1 22.8248,E2 188.1797} C_DIS
LIN {X -23.0924,Y -127.0166,Z 148,A -103.2784,B 22.8295,C -0.9511,E1 22.8186,E2 190.4354} C_DIS
LIN {X -27.015,Y -126.2401,Z 148,A -104.9302,B 22.8293,C -0.9574,E1 22.8141,E2 192.073} C_DIS
LIN {X -30.2297,Y -125.5089,Z 148,A -106.4163,B 22.8293,C -0.9572,E1 22.8101,E2 193.5619} C_DIS
LIN {X -33.9193,Y -124.5642,Z 148,A -108.1924,B 22.8294,C -0.9543,E1 22.8052,E2 195.3482} C_DIS
LIN {X -37.6267,Y -123.4931,Z 148,A -109.7425,B 22.8291,C -0.9629,E1 22.8011,E2 196.8792} C_DIS
LIN {X -40.5769,Y -122.5555,Z 148,A -111.1578,B 22.8291,C -0.9621,E1 22.7974,E2 198.2993} C_DIS
LIN {X -43.7086,Y -121.4737,Z 148,A -112.6263,B 22.8291,C -0.9635,E1 22.7935,E2 199.7675} C_DIS
LIN {X -46.6877,Y -120.3601,Z 148,A -113.8683,B 22.8287,C -0.9724,E1 22.7903,E2 200.9893} C_DIS
LIN {X -50.9473,Y -118.6202,Z 148,A -116.4018,B 22.8295,C -0.9526,E1 22.7836,E2 203.5801} C_DIS
LIN {X -55.4581,Y -116.5792,Z 148,A -118.2798,B 22.8288,C -0.9693,E1 22.779,E2 205.4202} C_DIS
LIN {X -58.2644,Y -115.2026,Z 148,A -119.6981,B 22.8288,C -0.9697,E1 22.7754,E2 206.8417} C_DIS
LIN {X -61.4915,Y -113.5152,Z 148,A -121.4273,B 22.8289,C -0.9668,E1 22.7711,E2 208.5837} C_DIS
LIN {X -65.142,Y -111.4601,Z 148,A -123.4921,B 22.8292,C -0.9605,E1 22.7661,E2 210.6717} C_DIS
LIN {X -67.9104,Y -109.7955,Z 148,A -124.4293,B 22.8282,C -0.9844,E1 22.764,E2 211.5502} C_DIS
LIN {X -70.7084,Y -108.0148,Z 148,A -126.229,B 22.8287,C -0.9723,E1 22.7597,E2 213.3876} C_DIS
LIN {X -73.0739,Y -106.4282,Z 148,A -127.8132,B 22.8292,C -0.9604,E1 22.756,E2 215.0084} C_DIS
LIN {X -76.264,Y -104.1662,Z 148,A -129.2269,B 22.8285,C -0.9774,E1 22.7528,E2 216.3837} C_DIS
LIN {X -79.9256,Y -101.384,Z 148,A -131.2444,B 22.8283,C -0.9821,E1 22.7484,E2 218.3971} C_DIS
LIN {X -83.2557,Y -98.668,Z 148,A -133.1863,B 22.8283,C -0.9842,E1 22.7442,E2 220.3418} C_DIS
LIN {X -86.5279,Y -95.8111,Z 148,A -135.1376,B 22.8281,C -0.9871,E1 22.7401,E2 222.2943} C_DIS
LIN {X -89.8229,Y -92.7286,Z 148,A -137.123,B 22.8279,C -0.992,E1 22.7361,E2 224.2762} C_DIS
LIN {X -93.0218,Y -89.5201,Z 148,A -139.1638,B 22.8278,C -0.995,E1 22.7321,E2 226.3188} C_DIS
LIN {X -95.394,Y -86.9875,Z 148,A -140.6911,B 22.8276,C -0.999,E1 22.7292,E2 227.8432} C_DIS
LIN {X -97.4213,Y -84.7106,Z 148,A -142.0289,B 22.8275,C -1.0027,E1 22.7268,E2 229.1779} C_DIS
LIN {X -100.2277,Y -81.3716,Z 148,A -143.7607,B 22.8269,C -1.016,E1 22.7237,E2 230.8841} C_DIS
LIN {X -103.1353,Y -77.6523,Z 148,A -146.0994,B 22.8271,C -1.0107,E1 22.7197,E2 233.249} C_DIS
LIN {X -105.6794,Y -74.1533,Z 148,A -148.0485,B 22.827,C -1.0142,E1 22.7165,E2 235.1995} C_DIS
LIN {X -108.155,Y -70.4933,Z 148,A -149.9873,B 22.8267,C -1.0202,E1 22.7135,E2 237.1334} C_DIS
LIN {X -110.3742,Y -66.9651,Z 148,A -151.7421,B 22.8263,C -1.0291,E1 22.711,E2 238.8751} C_DIS
LIN {X -112.7866,Y -62.8176,Z 148,A -154.3722,B 22.827,C -1.0137,E1 22.7073,E2 241.5604} C_DIS
LIN {X -114.6534,Y -59.3417,Z 148,A -155.8221,B 22.8263,C -1.0312,E1 22.7054,E2 242.9734} C_DIS
LIN {X -116.3913,Y -55.8513,Z 148,A -157.4439,B 22.8258,C -1.0407,E1 22.7035,E2 244.5803} C_DIS
LIN {X -117.8667,Y -52.6659,Z 148,A -158.9923,B 22.8256,C -1.0456,E1 22.7017,E2 246.1255} C_DIS
LIN {X -119.295,Y -49.3475,Z 148,A -160.6047,B 22.8255,C -1.0498,E1 22.6999,E2 247.7368} C_DIS
LIN {X -120.8316,Y -45.4537,Z 148,A -162.5807,B 22.8255,C -1.0503,E1 22.6979,E2 249.7239} C_DIS
LIN {X -122.7845,Y -39.8831,Z 148,A -165.1648,B 22.825,C -1.0596,E1 22.6956,E2 252.3001} C_DIS
LIN {X -123.8544,Y -36.4201,Z 148,A -166.4968,B 22.8243,C -1.0761,E1 22.6946,E2 253.5977} C_DIS
LIN {X -124.9559,Y -32.4475,Z 148,A -168.6738,B 22.8247,C -1.067,E1 22.6929,E2 255.8123} C_DIS
LIN {X -125.8582,Y -28.7408,Z 148,A -170.2777,B 22.8243,C -1.0761,E1 22.6919,E2 257.4032} C_DIS
LIN {X -126.5842,Y -25.3561,Z 148,A -171.959,B 22.8243,C -1.0748,E1 22.691,E2 259.0989} C_DIS
LIN {X -127.314,Y -21.3894,Z 148,A -173.6264,B 22.8239,C -1.0855,E1 22.6901,E2 260.7492} C_DIS
LIN {X -127.8355,Y -18.0143,Z 148,A -175.2239,B 22.8239,C -1.0869,E1 22.6895,E2 262.3538} C_DIS
LIN {X -128.3458,Y -13.9187,Z 148,A -176.9918,B 22.8234,C -1.0954,E1 22.6889,E2 264.1114} C_DIS
LIN {X -128.6706,Y -10.5062,Z 148,A -178.5918,B 22.8234,C -1.0969,E1 22.6885,E2 265.7179} C_DIS
LIN {X -128.934,Y -6.5119,Z 148,A 179.6416,B 22.8231,C -1.103,E1 22.6882,E2 267.4805} C_DIS
LIN {X -129.0601,Y -3.1712,Z 148,A 178.0266,B 22.8231,C -1.1023,E1 22.6882,E2 269.1081} C_DIS
LIN {X -129.0945,Y 1.1753,Z 148,A 176.2429,B 22.8225,C -1.1146,E1 22.6882,E2 270.8719} C_DIS
LIN {X -129.0075,Y 4.8476,Z 148,A 174.5802,B 22.8224,C -1.1185,E1 22.6882,E2 272.5355} C_DIS
LIN {X -128.8216,Y 8.465,Z 148,A 172.8533,B 22.8224,C -1.1187,E1 22.6885,E2 274.2733} C_DIS
LIN {X -128.4784,Y 12.6401,Z 148,A 171.021,B 22.822,C -1.1258,E1 22.689,E2 276.0993} C_DIS
LIN {X -128.0464,Y 16.4498,Z 148,A 169.4098,B 22.8216,C -1.1351,E1 22.6895,E2 277.6972} C_DIS
LIN {X -127.5699,Y 19.8059,Z 148,A 167.885,B 22.8214,C -1.1391,E1 22.6901,E2 279.2218} C_DIS
LIN {X -127.016,Y 23.0957,Z 148,A 166.3773,B 22.8212,C -1.1427,E1 22.6909,E2 280.73} C_DIS
LIN {X -126.2287,Y 27.0678,Z 148,A 164.5575,B 22.821,C -1.1475,E1 22.6919,E2 282.5492} C_DIS
LIN {X -125.4823,Y 30.3399,Z 148,A 163.0656,B 22.8208,C -1.1521,E1 22.6928,E2 284.0387} C_DIS
LIN {X -124.6396,Y 33.6367,Z 148,A 160.7352,B 22.8222,C -1.1229,E1 22.6946,E2 286.4599} C_DIS
LIN {X -123.0341,Y 39.1018,Z 148,A 158.9856,B 22.8203,C -1.1631,E1 22.696,E2 288.1166} C_DIS
LIN {X -122.0157,Y 42.1721,Z 148,A 157.6399,B 22.8199,C -1.1713,E1 22.6972,E2 289.4495} C_DIS
LIN {X -119.8938,Y 47.8741,Z 148,A 154.8053,B 22.8197,C -1.1739,E1 22.7,E2 292.2948} C_DIS
LIN {X -118.5635,Y 51.0782,Z 148,A 153.2988,B 22.8194,C -1.18,E1 22.7016,E2 293.7947} C_DIS
LIN {X -117.1785,Y 54.1799,Z 148,A 150.734,B 22.8213,C -1.1407,E1 22.7048,E2 296.4769} C_DIS
LIN {X -114.1499,Y 60.3005,Z 148,A 148.6801,B 22.8189,C -1.1901,E1 22.7073,E2 298.415} C_DIS
LIN {X -112.8573,Y 62.6898,Z 148,A 146.5637,B 22.8206,C -1.1557,E1 22.7103,E2 300.6329} C_DIS
LIN {X -109.6444,Y 68.1532,Z 148,A 144.6031,B 22.8185,C -1.1991,E1 22.713,E2 302.4921} C_DIS
LIN {X -107.354,Y 71.7068,Z 148,A 142.7045,B 22.8183,C -1.2034,E1 22.7159,E2 304.3901} C_DIS
LIN {X -105.4344,Y 74.5006,Z 148,A 140.8567,B 22.8188,C -1.1932,E1 22.7189,E2 306.2745} C_DIS
LIN {X -103.2352,Y 77.5199,Z 148,A 139.6507,B 22.8176,C -1.2166,E1 22.7208,E2 307.4263} C_DIS
LIN {X -100.1996,Y 81.4059,Z 148,A 137.277,B 22.8177,C -1.2145,E1 22.725,E2 309.8177} C_DIS
LIN {X -96.6315,Y 85.6103,Z 148,A 134.8974,B 22.8173,C -1.2236,E1 22.7293,E2 312.1855} C_DIS
LIN {X -93.8813,Y 88.6174,Z 148,A 133.0682,B 22.8171,C -1.2273,E1 22.7328,E2 314.0143} C_DIS
LIN {X -90.9892,Y 91.5844,Z 148,A 131.3913,B 22.8165,C -1.2386,E1 22.736,E2 315.6697} C_DIS
LIN {X -88.2144,Y 94.2607,Z 148,A 129.4125,B 22.8169,C -1.2312,E1 22.7401,E2 317.6767} C_DIS
LIN {X -84.6777,Y 97.45,Z 148,A 127.2386,B 22.8168,C -1.2335,E1 22.7446,E2 319.8543} C_DIS
LIN {X -80.9559,Y 100.5629,Z 148,A 125.4738,B 22.8157,C -1.2547,E1 22.7483,E2 321.5714} C_DIS
LIN {X -77.6955,Y 103.1027,Z 148,A 123.3667,B 22.8161,C -1.2469,E1 22.753,E2 323.7072} C_DIS
LIN {X -74.2221,Y 105.6309,Z 148,A 121.6683,B 22.8154,C -1.2597,E1 22.7568,E2 325.3791} C_DIS
LIN {X -71.5191,Y 107.4794,Z 148,A 119.9505,B 22.8158,C -1.2512,E1 22.7609,E2 327.1254} C_DIS
LIN {X -67.9947,Y 109.7431,Z 148,A 118.1769,B 22.8155,C -1.2583,E1 22.765,E2 328.8867} C_DIS
LIN {X -65.3203,Y 111.3554,Z 148,A 116.7641,B 22.8155,C -1.2597,E1 22.7684,E2 330.3008} C_DIS
LIN {X -59.7549,Y 114.4364,Z 148,A 113.9055,B 22.8152,C -1.2629,E1 22.7754,E2 333.1599} C_DIS
LIN {X -55.9489,Y 116.3447,Z 148,A 112.222,B 22.8146,C -1.2748,E1 22.7796,E2 334.8175} C_DIS
LIN {X -53.0738,Y 117.6843,Z 148,A 110.7568,B 22.8146,C -1.2745,E1 22.7833,E2 336.2877} C_DIS
LIN {X -49.9347,Y 119.0497,Z 148,A 109.1253,B 22.8148,C -1.2718,E1 22.7875,E2 337.9304} C_DIS
LIN {X -46.9366,Y 120.2633,Z 148,A 107.6954,B 22.8146,C -1.274,E1 22.7912,E2 339.3581} C_DIS
LIN {X -43.1881,Y 121.6613,Z 148,A 105.7212,B 22.815,C -1.2675,E1 22.7964,E2 341.3533} C_DIS
LIN {X -37.9282,Y 123.4009,Z 148,A 103.4342,B 22.8144,C -1.2779,E1 22.8025,E2 343.6181} C_DIS
LIN {X -34.8163,Y 124.3147,Z 148,A 101.9803,B 22.8144,C -1.2788,E1 22.8064,E2 345.0724} C_DIS
LIN {X -31.9144,Y 125.0912,Z 148,A 100.6238,B 22.8144,C -1.2791,E1 22.81,E2 346.4303} C_DIS
LIN {X -28.7083,Y 125.8657,Z 148,A 99.2031,B 22.8142,C -1.2823,E1 22.8139,E2 347.8447} C_DIS
LIN {X -25.5227,Y 126.5503,Z 148,A 97.7477,B 22.8142,C -1.2831,E1 22.8179,E2 349.3} C_DIS
LIN {X -19.5416,Y 127.6108,Z 148,A 95.0291,B 22.8142,C -1.284,E1 22.8254,E2 352.0192} C_DIS
LIN {X -14.9867,Y 128.2258,Z 148,A 93.1623,B 22.8136,C -1.2929,E1 22.8305,E2 353.8645} C_DIS
LIN {X -7.6022,Y 128.8748,Z 148,A 88.6925,B 22.8163,C -1.2421,E1 22.8433,E2 358.4673} C_DIS
LIN {X -0.93,Y 129.0953,Z 148,A 86.973,B 22.8134,C -1.2979,E1 22.8477,E2 360.043} C_DIS
LIN {X 5.4988,Y 128.9821,Z 148,A 83.0394,B 22.8159,C -1.2499,E1 22.859,E2 364.0994} C_DIS
LIN {X 11.3378,Y 128.6004,Z 148,A 81.4821,B 22.8135,C -1.2962,E1 22.863,E2 365.5364} C_DIS
LIN {X 17.3686,Y 127.926,Z 148,A 78.6549,B 22.8138,C -1.2896,E1 22.8709,E2 368.3785} C_DIS
LIN {X 20.221,Y 127.5056,Z 148,A 77.1733,B 22.8143,C -1.28,E1 22.875,E2 369.8832} C_DIS
LIN {X 23.9219,Y 126.8629,Z 148,A 75.6045,B 22.8141,C -1.2838,E1 22.8793,E2 371.4403} C_DIS
LIN {X 27.1929,Y 126.2017,Z 148,A 74.1666,B 22.8141,C -1.2851,E1 22.8832,E2 372.8729} C_DIS
LIN {X 30.8799,Y 125.3522,Z 148,A 72.364,B 22.8144,C -1.2785,E1 22.8882,E2 374.6898} C_DIS
LIN {X 34.6153,Y 124.3709,Z 148,A 70.7571,B 22.8142,C -1.2822,E1 22.8925,E2 376.2841} C_DIS
LIN {X 37.8451,Y 123.4263,Z 148,A 69.2977,B 22.8142,C -1.2827,E1 22.8964,E2 377.7396} C_DIS
LIN {X 40.9285,Y 122.4384,Z 148,A 67.8349,B 22.8143,C -1.2803,E1 22.9002,E2 379.2054} C_DIS
LIN {X 44.7084,Y 121.1108,Z 148,A 65.7212,B 22.8152,C -1.2632,E1 22.9059,E2 381.3582} C_DIS
LIN {X 47.8616,Y 119.8988,Z 148,A 64.7341,B 22.814,C -1.2853,E1 22.9083,E2 382.2861} C_DIS
LIN {X 51.6702,Y 118.3076,Z 148,A 62.6555,B 22.8148,C -1.2718,E1 22.9137,E2 384.3939} C_DIS
LIN {X 55.2989,Y 116.6552,Z 148,A 60.9562,B 22.8148,C -1.273,E1 22.918,E2 386.0854} C_DIS
LIN {X 58.2036,Y 115.2335,Z 148,A 59.4722,B 22.8149,C -1.2689,E1 22.9217,E2 387.5755} C_DIS
LIN {X 61.6588,Y 113.4239,Z 148,A 57.8171,B 22.8149,C -1.27,E1 22.9258,E2 389.2224} C_DIS
LIN {X 65.3348,Y 111.3468,Z 148,A 55.9674,B 22.8149,C -1.2684,E1 22.9303,E2 391.07} C_DIS
LIN {X 68.6059,Y 109.3623,Z 148,A 54.1519,B 22.8154,C -1.2603,E1 22.9346,E2 392.9} C_DIS
LIN {X 72.0595,Y 107.1183,Z 148,A 52.3061,B 22.8156,C -1.2565,E1 22.9389,E2 394.7489} C_DIS
LIN {X 75.7606,Y 104.5327,Z 148,A 50.3556,B 22.8156,C -1.2556,E1 22.9433,E2 396.6943} C_DIS
LIN {X 79.3518,Y 101.8339,Z 148,A 48.3829,B 22.8158,C -1.2529,E1 22.9477,E2 398.6658} C_DIS
LIN {X 82.6005,Y 99.217,Z 148,A 46.5155,B 22.816,C -1.2486,E1 22.9518,E2 400.5364} C_DIS
LIN {X 85.8585,Y 96.4116,Z 148,A 44.6267,B 22.8161,C -1.2458,E1 22.9557,E2 402.4243} C_DIS
LIN {X 89.0808,Y 93.4416,Z 148,A 42.6369,B 22.8164,C -1.2396,E1 22.9598,E2 404.4208} C_DIS
LIN {X 91.2884,Y 91.2872,Z 148,A 41.2886,B 22.8165,C -1.2376,E1 22.9625,E2 405.768} C_DIS
LIN {X 95.3657,Y 87.0188,Z 148,A 38.6986,B 22.8168,C -1.2332,E1 22.9674,E2 408.3568} C_DIS
LIN {X 98.1955,Y 83.812,Z 148,A 36.8055,B 22.817,C -1.2291,E1 22.9709,E2 410.2511} C_DIS
LIN {X 101.1666,Y 80.2006,Z 148,A 34.7814,B 22.8171,C -1.2265,E1 22.9744,E2 412.2712} C_DIS
LIN {X 103.7562,Y 76.8214,Z 148,A 32.8656,B 22.8174,C -1.2206,E1 22.9777,E2 414.1921} C_DIS
LIN {X 106.2474,Y 73.3373,Z 148,A 30.999,B 22.8176,C -1.2174,E1 22.9807,E2 416.0567} C_DIS
LIN {X 108.5874,Y 69.8255,Z 148,A 29.284,B 22.8174,C -1.2202,E1 22.9833,E2 417.7553} C_DIS
LIN {X 109.913,Y 67.7188,Z 148,A 27.6721,B 22.8188,C -1.1929,E1 22.9857,E2 419.428} C_DIS
LIN {X 111.9861,Y 64.2337,Z 148,A 26.2178,B 22.8182,C -1.2046,E1 22.9877,E2 420.844} C_DIS
LIN {X 114.1128,Y 60.3712,Z 148,A 24.376,B 22.8182,C -1.2048,E1 22.9901,E2 422.6746} C_DIS
LIN {X 115.6641,Y 57.3422,Z 148,A 23.0006,B 22.8181,C -1.2071,E1 22.9918,E2 424.0361} C_DIS
LIN {X 117.4035,Y 53.6933,Z 148,A 21.1235,B 22.8185,C -1.198,E1 22.9941,E2 425.9254} C_DIS
LIN {X 118.9454,Y 50.1844,Z 148,A 19.1179,B 22.8195,C -1.1783,E1 22.9963,E2 427.9691} C_DIS
LIN {X 120.1689,Y 47.1796,Z 148,A 18.0405,B 22.8189,C -1.1916,E1 22.9974,E2 429.0059} C_DIS
LIN {X 121.4372,Y 43.8097,Z 148,A 16.4235,B 22.8191,C -1.186,E1 22.999,E2 430.6273} C_DIS
LIN {X 122.5086,Y 40.7177,Z 148,A 14.9589,B 22.8194,C -1.181,E1 23.0003,E2 432.0954} C_DIS
LIN {X 123.6679,Y 37.0556,Z 148,A 13.198,B 22.8198,C -1.1731,E1 23.0017,E2 433.8655} C_DIS
LIN {X 124.6367,Y 33.6477,Z 148,A 11.6852,B 22.8198,C -1.1712,E1 23.0029,E2 435.3736} C_DIS
LIN {X 125.4813,Y 30.3443,Z 148,A 10.2417,B 22.8199,C -1.17,E1 23.0038,E2 436.8112} C_DIS
LIN {X 126.1779,Y 27.3034,Z 148,A 8.9952,B 22.8199,C -1.1724,E1 23.0046,E2 438.0434} C_DIS
LIN {X 126.8786,Y 23.8394,Z 148,A 7.1507,B 22.8207,C -1.154,E1 23.0056,E2 439.9231} C_DIS
LIN {X 128.1341,Y 15.7556,Z 148,A 3.8214,B 22.8205,C -1.1572,E1 23.007,E2 443.2225} C_DIS
LIN {X 128.7389,Y 9.6291,Z 148,A 0.9278,B 22.8213,C -1.1406,E1 23.0077,E2 446.1398} C_DIS
LIN {X 128.9731,Y 5.7272,Z 148,A -0.9014,B 22.8218,C -1.1303,E1 23.008,E2 447.9832} C_DIS
LIN {X 129.0924,Y 1.4353,Z 148,A -3.2661,B 22.8231,C -1.1019,E1 23.008,E2 450.4051} C_DIS
LIN {X 129.0573,Y -3.2727,Z 148,A -4.7341,B 22.822,C -1.1254,E1 23.008,E2 451.8033} C_DIS
LIN {X 128.6843,Y -10.3442,Z 148,A -7.8517,B 22.8225,C -1.1164,E1 23.0075,E2 454.9235} C_DIS
LIN {X 127.8825,Y -17.6853,Z 148,A -11.0933,B 22.8229,C -1.1075,E1 23.0065,E2 458.1666} C_DIS
LIN {X 126.8223,Y -24.1339,Z 148,A -14.0737,B 22.8235,C -1.0943,E1 23.005,E2 461.1615} C_DIS
LIN {X 125.9024,Y -28.5473,Z 148,A -15.9154,B 22.8235,C -1.0957,E1 23.004,E2 462.9878} C_DIS
LIN {X 125.1488,Y -31.6877,Z 148,A -17.409,B 22.8238,C -1.0882,E1 23.003,E2 464.4911} C_DIS
LIN {X 124.2638,Y -34.9983,Z 148,A -18.9179,B 22.8239,C -1.0839,E1 23.0018,E2 466.0013} C_DIS
LIN {X 123.0965,Y -38.9063,Z 148,A -20.7545,B 22.8243,C -1.077,E1 23.0003,E2 467.8442} C_DIS
LIN {X 121.9755,Y -42.2878,Z 148,A -22.2641,B 22.8243,C -1.0755,E1 22.999,E2 469.3481} C_DIS
LIN {X 120.7994,Y -45.5398,Z 148,A -23.6794,B 22.8243,C -1.0766,E1 22.9976,E2 470.7518} C_DIS
LIN {X 119.8862,Y -47.893,Z 148,A -25.0035,B 22.8249,C -1.0632,E1 22.9963,E2 472.1022} C_DIS
LIN {X 118.3821,Y -51.4978,Z 148,A -26.6522,B 22.8249,C -1.062,E1 22.9945,E2 473.7439} C_DIS
LIN {X 116.1436,Y -56.3653,Z 148,A -29.2593,B 22.8257,C -1.0437,E1 22.9913,E2 476.3823} C_DIS
LIN {X 114.7057,Y -59.2405,Z 148,A -30.5434,B 22.8257,C -1.0464,E1 22.9897,E2 477.6521} C_DIS
LIN {X 112.5577,Y -63.226,Z 148,A -32.4106,B 22.8256,C -1.0474,E1 22.9872,E2 479.5059} C_DIS
LIN {X 109.843,Y -67.8337,Z 148,A -34.7727,B 22.8258,C -1.0411,E1 22.9838,E2 481.8707} C_DIS
LIN {X 107.2788,Y -71.8194,Z 148,A -36.937,B 22.8262,C -1.0322,E1 22.9805,E2 484.0458} C_DIS
LIN {X 104.7978,Y -75.3944,Z 148,A -38.783,B 22.8262,C -1.0311,E1 22.9775,E2 485.8849} C_DIS
LIN {X 100.0425,Y -81.5982,Z 148,A -42.3941,B 22.8269,C -1.0149,E1 22.9713,E2 489.5186} C_DIS
LIN {X 96.5328,Y -85.7217,Z 148,A -44.9635,B 22.8275,C -1.0007,E1 22.9665,E2 492.1116} C_DIS
LIN {X 94.1472,Y -88.3356,Z 148,A -46.0334,B 22.8267,C -1.0209,E1 22.9646,E2 493.1245} C_DIS
LIN {X 89.536,Y -93.0064,Z 148,A -49.1531,B 22.8274,C -1.0038,E1 22.9584,E2 496.2734} C_DIS
LIN {X 87.0128,Y -95.3711,Z 148,A -50.8125,B 22.8278,C -0.9942,E1 22.955,E2 497.95} C_DIS
LIN {X 83.6405,Y -98.3413,Z 148,A -53.3138,B 22.829,C -0.9655,E1 22.9495,E2 500.5141} C_DIS
LIN {X 79.3983,Y -101.798,Z 148,A -55.0749,B 22.8279,C -0.992,E1 22.9458,E2 502.1999} C_DIS
LIN {X 77.0333,Y -103.5984,Z 148,A -56.6307,B 22.8285,C -0.9779,E1 22.9423,E2 503.7857} C_DIS
LIN {X 74.3111,Y -105.5681,Z 148,A -58.3004,B 22.8289,C -0.9664,E1 22.9384,E2 505.4786} C_DIS
LIN {X 70.7441,Y -107.9912,Z 148,A -59.7548,B 22.8282,C -0.9845,E1 22.9351,E2 506.8812} C_DIS
LIN {X 66.3254,Y -110.7596,Z 148,A -62.7035,B 22.8296,C -0.9502,E1 22.9279,E2 509.9078} C_DIS
LIN {X 61.7447,Y -113.377,Z 148,A -64.1551,B 22.8281,C -0.9882,E1 22.9246,E2 511.2571} C_DIS
LIN {X 59.0349,Y -114.8103,Z 148,A -65.7539,B 22.8286,C -0.9746,E1 22.9206,E2 512.886} C_DIS
LIN {X 55.8493,Y -116.3923,Z 148,A -67.284,B 22.8286,C -0.9743,E1 22.9168,E2 514.4122} C_DIS
LIN {X 53.1834,Y -117.6353,Z 148,A -68.6739,B 22.8289,C -0.9683,E1 22.9132,E2 515.8137} C_DIS
LIN {X 47.0642,Y -120.2135,Z 148,A -71.567,B 22.8289,C -0.9667,E1 22.9057,E2 518.7036} C_DIS
LIN {X 43.7371,Y -121.4634,Z 148,A -73.9149,B 22.8304,C -0.9286,E1 22.8993,E2 521.144} C_DIS
LIN {X 38.0555,Y -123.3619,Z 148,A -75.7452,B 22.829,C -0.964,E1 22.8947,E2 522.8795} C_DIS
LIN {X 34.8309,Y -124.3106,Z 148,A -77.2033,B 22.829,C -0.964,E1 22.8908,E2 524.3349} C_DIS
LIN {X 31.7463,Y -125.1339,Z 148,A -78.618,B 22.829,C -0.9626,E1 22.887,E2 525.7507} C_DIS
LIN {X 27.7496,Y -126.0815,Z 148,A -80.5286,B 22.8293,C -0.9568,E1 22.8817,E2 527.6734} C_DIS
LIN {X 23.3931,Y -126.9627,Z 148,A -83.2309,B 22.8307,C -0.9215,E1 22.8741,E2 530.463} C_DIS
LIN {X 17.6253,Y -127.891,Z 148,A -84.844,B 22.829,C -0.9649,E1 22.8699,E2 531.9628} C_DIS
LIN {X 11.6886,Y -128.5697,Z 148,A -87.7678,B 22.8296,C -0.9508,E1 22.8617,E2 534.9208} C_DIS
LIN {X 4.2536,Y -129.03,Z 148,A -90.8982,B 22.8293,C -0.9576,E1 22.8531,E2 538.0324} C_DIS
LIN {X 0.9253,Y -129.0761,Z 148,A -92.2766,B 22.8291,C -0.9621,E1 22.8493,E2 539.399} C_DIS
Enddeposition()
LIN {X 0.9253,Y -129.0761,Z 148,A -92.2766,B 22.8291,C -0.9621,E1 22.8493,E2 539.399} C_DIS
Startdeposition()
$VEL.CP = VEL_PRINT
LIN {X 4.5902,Y -128.0648,Z 148,A -89.0261,B 21.8602,C -0.8771,E1 21.8867,E2 536.2545} C_DIS
LIN {X 10.2958,Y -127.733,Z 148,A -87.3661,B 21.8617,C -0.8382,E1 21.891,E2 534.6999} C_DIS
LIN {X 17.2672,Y -126.9791,Z 148,A -84.0538,B 21.8613,C -0.8478,E1 21.9002,E2 531.3647} C_DIS
LIN {X 23.2554,Y -126.0203,Z 148,A -81.3641,B 21.8613,C -0.8488,E1 21.9076,E2 528.6756} C_DIS
LIN {X 26.7301,Y -125.3277,Z 148,A -79.879,B 21.8613,C -0.8457,E1 21.9117,E2 527.2009} C_DIS
LIN {X 30.7791,Y -124.397,Z 148,A -77.8608,B 21.8611,C -0.8547,E1 21.9172,E2 525.162} C_DIS
LIN {X 34.6123,Y -123.3832,Z 148,A -76.1878,B 21.8611,C -0.852,E1 21.9217,E2 523.4992} C_DIS
LIN {X 38.6495,Y -122.1792,Z 148,A -73.4647,B 21.8596,C -0.8924,E1 21.9292,E2 520.6736} C_DIS
LIN {X 44.4899,Y -120.176,Z 148,A -71.5451,B 21.861,C -0.8575,E1 21.934,E2 518.8522} C_DIS
LIN {X 47.0717,Y -119.1894,Z 148,A -69.9712,B 21.8603,C -0.8746,E1 21.9382,E2 517.2367} C_DIS
LIN {X 50.4213,Y -117.8104,Z 148,A -68.3971,B 21.8603,C -0.8749,E1 21.9422,E2 515.6662} C_DIS
LIN {X 53.5682,Y -116.4125,Z 148,A -67.2217,B 21.8608,C -0.8605,E1 21.9451,E2 514.5326} C_DIS
LIN {X 56.556,Y -114.9904,Z 148,A -65.7124,B 21.8608,C -0.8642,E1 21.9489,E2 513.018} C_DIS
LIN {X 59.2467,Y -113.628,Z 148,A -64.5486,B 21.8609,C -0.858,E1 21.9517,E2 511.8745} C_DIS
LIN {X 61.9567,Y -112.1751,Z 148,A -62.8693,B 21.8603,C -0.8743,E1 21.9559,E2 510.1573} C_DIS
LIN {X 68.0716,Y -108.5738,Z 148,A -59.777,B 21.8603,C -0.8763,E1 21.9633,E2 507.0707} C_DIS
LIN {X 71.5748,Y -106.2968,Z 148,A -57.7217,B 21.8598,C -0.8886,E1 21.9682,E2 504.9905} C_DIS
LIN {X 78.0112,Y -101.6669,Z 148,A -54.4066,B 21.8599,C -0.8852,E1 21.9756,E2 501.6982} C_DIS
LIN {X 80.5925,Y -99.633,Z 148,A -52.427,B 21.8589,C -0.9122,E1 21.98,E2 499.6553} C_DIS
LIN {X 84.1932,Y -96.6094,Z 148,A -50.1064,B 21.8583,C -0.9272,E1 21.9849,E2 497.3052} C_DIS
LIN {X 88.5238,Y -92.6574,Z 148,A -48.4285,B 21.8598,C -0.8892,E1 21.9881,E2 495.7368} C_DIS
LIN {X 93.6855,Y -87.4351,Z 148,A -44.483,B 21.8582,C -0.9281,E1 21.9959,E2 491.7072} C_DIS
LIN {X 96.789,Y -83.9874,Z 148,A -42.9001,B 21.8589,C -0.9103,E1 21.9988,E2 490.18} C_DIS
LIN {X 99.3016,Y -81.0003,Z 148,A -40.5199,B 21.8575,C -0.9447,E1 22.0031,E2 487.7207} C_DIS
LIN {X 102.6639,Y -76.6943,Z 148,A -38.7608,B 21.8586,C -0.919,E1 22.0059,E2 486.04} C_DIS
LIN {X 105.0722,Y -73.3604,Z 148,A -36.9485,B 21.8584,C -0.9228,E1 22.0089,E2 484.2279} C_DIS
LIN {X 107.0134,Y -70.4981,Z 148,A -35.0874,B 21.8577,C -0.9419,E1 22.0118,E2 482.3265} C_DIS
LIN {X 109.0008,Y -67.3857,Z 148,A -34.0146,B 21.8586,C -0.9193,E1 22.0133,E2 481.3202} C_DIS
LIN {X 111.2761,Y -63.5571,Z 148,A -31.7741,B 21.8579,C -0.9367,E1 22.0165,E2 479.0467} C_DIS
LIN {X 113.321,Y -59.8313,Z 148,A -30.1934,B 21.8583,C -0.9273,E1 22.0185,E2 477.5008} C_DIS
LIN {X 115.1427,Y -56.2474,Z 148,A -28.0851,B 21.8574,C -0.9471,E1 22.0212,E2 475.3525} C_DIS
LIN {X 116.8723,Y -52.5577,Z 148,A -26.4039,B 21.8574,C -0.9459,E1 22.0232,E2 473.685} C_DIS
LIN {X 118.1145,Y -49.7038,Z 148,A -25.0405,B 21.8574,C -0.9488,E1 22.0247,E2 472.3227} C_DIS
LIN {X 119.349,Y -46.6612,Z 148,A -23.3674,B 21.8568,C -0.963,E1 22.0264,E2 470.6226} C_DIS
LIN {X 120.9946,Y -42.2109,Z 148,A -21.4273,B 21.8568,C -0.9609,E1 22.0282,E2 468.7006} C_DIS
LIN {X 122.0266,Y -39.127,Z 148,A -19.9463,B 21.8566,C -0.9667,E1 22.0295,E2 467.2138} C_DIS
LIN {X 123.1959,Y -35.281,Z 148,A -18.1072,B 21.8563,C -0.9742,E1 22.031,E2 465.3668} C_DIS
LIN {X 124.1867,Y -31.6086,Z 148,A -16.5262,B 21.8563,C -0.974,E1 22.0321,E2 463.7971} C_DIS
LIN {X 125.0025,Y -28.2121,Z 148,A -14.9057,B 21.856,C -0.9817,E1 22.0331,E2 462.1669} C_DIS
LIN {X 125.867,Y -24.061,Z 148,A -12.2911,B 21.8542,C -1.0218,E1 22.0346,E2 459.4629} C_DIS
LIN {X 126.8155,Y -18.422,Z 148,A -10.5423,B 21.8556,C -0.9916,E1 22.0353,E2 457.8067} C_DIS
LIN {X 127.6933,Y -10.7664,Z 148,A -7.4718,B 21.8559,C -0.9849,E1 22.0362,E2 454.7751} C_DIS
LIN {X 128.0814,Y -4.1185,Z 148,A -4.2868,B 21.855,C -1.0041,E1 22.0367,E2 451.5609} C_DIS
LIN {X 128.1215,Y 2.5652,Z 148,A -0.9344,B 21.8538,C -1.0308,E1 22.0367,E2 448.1606} C_DIS
LIN {X 127.9401,Y 7.2912,Z 148,A 0.9836,B 21.854,C -1.0282,E1 22.0364,E2 446.2626} C_DIS
LIN {X 127.1977,Y 15.5677,Z 148,A 4.509,B 21.8538,C -1.0309,E1 22.0355,E2 442.7541} C_DIS
LIN {X 126.5159,Y 20.388,Z 148,A 6.8729,B 21.8531,C -1.0465,E1 22.0345,E2 440.3647} C_DIS
LIN {X 125.8415,Y 24.1948,Z 148,A 8.4434,B 21.8532,C -1.0445,E1 22.0337,E2 438.8103} C_DIS
LIN {X 125.0947,Y 27.8082,Z 148,A 10.2279,B 21.8527,C -1.0559,E1 22.0326,E2 437.0075} C_DIS
LIN {X 124.2304,Y 31.4361,Z 148,A 11.7003,B 21.8529,C -1.0519,E1 22.0316,E2 435.5556} C_DIS
LIN {X 123.4422,Y 34.4013,Z 148,A 13.0699,B 21.8527,C -1.0559,E1 22.0306,E2 434.1843} C_DIS
LIN {X 122.5726,Y 37.3815,Z 148,A 14.474,B 21.8525,C -1.0609,E1 22.0295,E2 432.7764} C_DIS
LIN {X 121.5971,Y 40.442,Z 148,A 15.9023,B 21.8523,C -1.0648,E1 22.0283,E2 431.3469} C_DIS
LIN {X 120.4465,Y 43.7508,Z 148,A 17.4166,B 21.8522,C -1.067,E1 22.0269,E2 429.8367} C_DIS
LIN {X 119.3501,Y 46.6583,Z 148,A 18.8027,B 21.852,C -1.0709,E1 22.0255,E2 428.4491} C_DIS
LIN {X 117.3373,Y 51.5154,Z 148,A 21.2501,B 21.8515,C -1.0821,E1 22.0228,E2 425.9873} C_DIS
LIN {X 115.857,Y 54.7613,Z 148,A 22.931,B 21.8511,C -1.0906,E1 22.0208,E2 424.2942} C_DIS
LIN {X 113.7829,Y 58.9517,Z 148,A 24.9463,B 21.851,C -1.0929,E1 22.0183,E2 422.2854} C_DIS
LIN {X 111.7773,Y 62.6715,Z 148,A 26.7488,B 21.851,C -1.094,E1 22.0158,E2 420.4909} C_DIS
LIN {X 109.8122,Y 66.0547,Z 148,A 28.5718,B 21.8505,C -1.102,E1 22.0132,E2 418.6571} C_DIS
LIN {X 107.5527,Y 69.6728,Z 148,A 30.3862,B 21.8505,C -1.1027,E1 22.0105,E2 416.8517} C_DIS
LIN {X 105.3047,Y 73.0261,Z 148,A 32.2552,B 21.8501,C -1.1102,E1 22.0076,E2 414.9731} C_DIS
LIN {X 102.6057,Y 76.7725,Z 148,A 34.263,B 21.8501,C -1.1127,E1 22.0043,E2 412.97} C_DIS
LIN {X 100.0273,Y 80.1033,Z 148,A 36.206,B 21.8497,C -1.12,E1 22.0009,E2 411.0181} C_DIS
LIN {X 97.2096,Y 83.4996,Z 148,A 38.1193,B 21.8496,C -1.1219,E1 21.9975,E2 409.11} C_DIS
LIN {X 94.3923,Y 86.6715,Z 148,A 39.7522,B 21.85,C -1.114,E1 21.9945,E2 407.5064} C_DIS
LIN {X 91.1268,Y 90.0992,Z 148,A 41.9585,B 21.8495,C -1.1227,E1 21.9902,E2 405.288} C_DIS
Enddeposition()
END
